// TIA Portal project "paletizer_2026_03_07" (V18)
// Vorlageprojekt für das Buch mit Zielsystem S7-1200

(* hardware
DEVICE "S7-1200 station_1"  S7-1200 Station
   slot 0: "Rack_0"  S7-1200 Rack  Rack  V1.0
   slot 1: "PLC_2"  CPU 1215C DC/DC/DC  6ES7 215-1AG40-0XB0  V4.4
   slot 2: "DI 16/DQ 16x24VDC_1"  6ES7 223-1BL32-0XB0  V2.0
   slot 3: "DI 16x24VDC_1"  6ES7 221-1BH32-0XB0  V2.0
   slot 4: "AI 4x13BIT/AQ 2x14BIT_1"  6ES7 234-4HE32-0XB0  V2.1
DEVICE "HMI_1"  KTP1200 Basic PN
   slot 0: "HMI_1"  KTP1200 Basic PN  6AV2 123-2MB03-0AX0  17.0.0.0
   slot 1: "HMI_RT_1"  KTP1200 Basic PN  6AV2 123-2MB03-0AX0  17.0.0.0
   slot 5: "HMI_1.IE_CP_1"  PROFINET Interface  17.0.0.0
      slot 1: "PROFINET Interface_1"  PROFINET Interface
         slot 1: "Port_1"  Port
*)

// ===== PLC "PLC_2"  CPU 1215C DC/DC/DC =====

VAR_GLOBAL   // PLC tag table "Default tag table"
   "Security Relay" AT %I10.0 : Bool;
   "Emergency stop feeding" AT %I10.1 : Bool;
   "Emergency stop elevator" AT %I10.2 : Bool;
   "Emergency stop load beld" AT %I10.3 : Bool;
   "Select auto" AT %I10.4 : Bool;
   "Select manual" AT %I10.5 : Bool;
   "Fault reset button" AT %I10.6 : Bool;
   "Manual box feeding button" AT %I11.0 : Bool;
   "Manual load beld" AT %I11.1 : Bool;
   "Manual Clamp" AT %I11.2 : Bool;
   "Box feeder motor guard" AT %I12.0 : Bool;
   "Enable load beld motor guard" AT %I12.1 : Bool;
   "Elevator motor guard" AT %I12.2 : Bool;
   "Load pallet motor guard" AT %I12.3 : Bool;
   "Pallet feeder motor guard" AT %I12.4 : Bool;
   "Exit conveyor motor guard" AT %I12.5 : Bool;
   "Box feeder motor feedback" AT %I13.0 : Bool;
   "Enable load beld motor feedback" AT %I13.1 : Bool;
   "Elevator motor feedback up" AT %I13.2 : Bool;
   "Elevator motor feedback down" AT %I13.3 : Bool;
   "Load pallet motor feedback" AT %I13.4 : Bool;
   "Pallet feeder motor feedback" AT %I13.5 : Bool;
   "Exit conveyor motor feedback" AT %I13.6 : Bool;
   "Pallet at entry" AT %I14.0 : Bool;
   "Pallet at exit" AT %I14.1 : Bool;
   "Pallet loaded" AT %I14.2 : Bool;
   "Up load pallet" AT %I14.3 : Bool;
   "Down load pallet" AT %I14.4 : Bool;
   "Box at entry" AT %I14.5 : Bool;
   "Pusher limit" AT %I14.6 : Bool;
   "Plate limit" AT %I14.7 : Bool;
   "Clamped" AT %I15.0 : Bool;
   "Manual pallet feeder" AT %I11.3 : Bool;
   "Manual load pallet" AT %I11.4 : Bool;
   "Elevator moving" AT %I15.1 : Bool;
   "Manual exit conveyor" AT %I11.5 : Bool;
   "Manual elevator up" AT %I15.2 : Bool;
   "Manual elevator down" AT %I15.3 : Bool;
   "Relay warning ligth" AT %Q10.0 : Bool;
   "Relay aux turn valve" AT %Q10.1 : Bool;
   "Relay aux push valve" AT %Q10.2 : Bool;
   "Relay aux plate valve" AT %Q10.3 : Bool;
   "Relay Clamp" AT %Q10.4 : Bool;
   "Move to limit" AT %Q10.5 : Bool;
   "Enable pallet emiter" AT %Q10.6 : Bool;
   "Enable exit conveyor" AT %Q10.7 : Bool;
   "Enable box feeder motor" AT %Q12.0 : Bool;
   "Enable load beld motor" AT %Q12.1 : Bool;
   "Enable elevator up motor" AT %Q12.2 : Bool;
   "Enable elevator down motor" AT %Q12.3 : Bool;
   "Enable Load pallet motor" AT %Q12.4 : Bool;
   "Enable Pallet feeder motor" AT %Q12.5 : Bool;
   "Enable exit conveyor motor" AT %Q12.6 : Bool;
   "Fault reset light" AT %Q13.0 : Bool;
   "Start feeding light" AT %Q13.1 : Bool;
   "Stop feeding light" AT %Q13.2 : Bool;
   "Counter box" AT %QW50 : Word;
   "Input_Security_Relay" AT %M0.0 : Bool;
   "Input_Emergency_stop_feeding" AT %M0.1 : Bool;
   "Input_emergency_stop_elevator" AT %M0.2 : Bool;
   "Input_emergency_stop_load_beld" AT %M0.3 : Bool;
   "Input_select_auto" AT %M0.4 : Bool;
   "Input_select_manual" AT %M0.5 : Bool;
   "Input_Fault_reset_button" AT %M0.6 : Bool;
   "Input_manual_box_feeding_button" AT %M1.0 : Bool;
   "Input_manual_load_beld" AT %M1.1 : Bool;
   "Input_manual_clamp" AT %M1.2 : Bool;
   "Input_manual_pallet_feeder" AT %M1.3 : Bool;
   "Input_box_feeder_motor_guard" AT %M2.0 : Bool;
   "Input_enable_load_beld_motor_guard" AT %M2.1 : Bool;
   "Input_elevator_motor_guard" AT %M2.2 : Bool;
   "Input_load_pallet_motor_guard" AT %M2.3 : Bool;
   "Input_pallet_feeder_motor_guad" AT %M2.4 : Bool;
   "Input_box_feeder_motor_feedback" AT %M3.0 : Bool;
   "Input_enable_load_beld_motor_feedback" AT %M3.1 : Bool;
   "Input_elevator_motor_feedback_up" AT %M3.2 : Bool;
   "Input_elevator_motor_feedback_down" AT %M3.3 : Bool;
   "Input_load_pallet_motor_feedback" AT %M3.4 : Bool;
   "Input_pallet_feeder_motor_feedback" AT %M3.5 : Bool;
   "Input_pallet_at_entry" AT %M4.0 : Bool;
   "Input_pallet_at_exit" AT %M4.1 : Bool;
   "Input_pallet_loaded" AT %M4.2 : Bool;
   "Input_up_load_pallet" AT %M4.3 : Bool;
   "Input_down_load_pallet" AT %M4.4 : Bool;
   "Input_box_at_entry" AT %M4.5 : Bool;
   "Input_pusher_limit" AT %M4.6 : Bool;
   "Input_plate_limit" AT %M4.7 : Bool;
   "Input_clamped" AT %M5.0 : Bool;
   "Output_warning_ligth" AT %M10.0 : Bool;
   "Output_relay_aux_turn_valve" AT %M10.1 : Bool;
   "Ouput_relay_aux_push_valve" AT %M10.2 : Bool;
   "Output_relay_aux_plate_valve" AT %M10.3 : Bool;
   "Output_relay_clamp" AT %M10.4 : Bool;
   "Ouput_move_to_limit" AT %M10.5 : Bool;
   "Output_enable_pallet_emiter" AT %M10.6 : Bool;
   "Output_enable_exit_conveyor" AT %M10.7 : Bool;
   "Output_enable_box_feeder_motor" AT %M12.0 : Bool;
   "Output_enable_load_beld_motor" AT %M12.1 : Bool;
   "Output_enable_elevator_up_motor" AT %M12.2 : Bool;
   "Output_enable_elevator_down_motor" AT %M12.3 : Bool;
   "Output_enable_load_pallet_motor" AT %M12.4 : Bool;
   "Output_enable_pallet_feeder_motor" AT %M12.5 : Bool;
   "Output_enable_exit_conveyor_motor" AT %M12.6 : Bool;
   "Output_fault_reset_light" AT %M13.0 : Bool;
   "Output_start_feeding_light" AT %M13.1 : Bool;
   "Output_stop_feeding_light" AT %M13.2 : Bool;
   "Ouput_counter_box" AT %MW100 : Word;
   "Emergency_enable" AT %M30.0 : Bool;
   "Manual_box_feeding_drive" AT %M30.1 : Bool;
   "Input_manual_load_pallet" AT %M1.4 : Bool;
   "Input_manual_exit_conveyor" AT %M1.5 : Bool;
   "Manual_load_beld_drive" AT %M30.2 : Bool;
   "Manual_clamp_drive" AT %M30.3 : Bool;
   "Manual_pallet_feeder_drive" AT %M30.4 : Bool;
   "Input_elevator_moving" AT %M5.1 : Bool;
   "Input_manual_elevator_up" AT %M5.2 : Bool;
   "Input_manual_elevator_down" AT %M5.3 : Bool;
   "Manual_load_pallet_drive" AT %M30.5 : Bool;
   "Manual_exit_conveyor_drive" AT %M30.6 : Bool;
   "Manual_elevator_up_drive" AT %M30.7 : Bool;
   "Manual_elevator_down_drive" AT %M31.0 : Bool;
   "Input_exit_conveyor_motor_guard" AT %M2.5 : Bool;
   "Input_exit_conveyor_motor_feedback" AT %M3.6 : Bool;
   "Aux_manual_box_feeding_drive" AT %M31.1 : Bool;
   "Up_manual_box_feeding_drive" AT %M6.0 : Bool;
   "Up_manual_load_beld_drive" AT %M6.1 : Bool;
   "Aux_manual_load_beld_drive" AT %M31.2 : Bool;
   "Aux_manual_pallet_feeder_drive" AT %M31.4 : Bool;
   "Aux_manual_load_pallet_drive" AT %M31.5 : Bool;
   "Aux_manual_exit_conveyor_drive" AT %M31.6 : Bool;
   "Aux_manual_elevator_up_drive" AT %M31.7 : Bool;
   "Aux_manual_elevator_down_drive" AT %M32.0 : Bool;
   "Up_manual_pallet_feeder_drive" AT %M6.2 : Bool;
   "Up_manual_load_pallet_drive" AT %M6.3 : Bool;
   "Up_manual_exit_conveyor_drive" AT %M6.4 : Bool;
   "Up_manual_elevator_up_drive" AT %M6.5 : Bool;
   "Up_manual_elevator_down_drive" AT %M6.6 : Bool;
   "Zero_Point" AT %M15.0 : Bool;
   "Reset_value_counters" AT %M15.2 : Bool;
   "Enable_Box_Feeder_Auto" AT %M15.3 : Bool;
   "Enable_Turn_Auto" AT %M15.4 : Bool;
   "Enable_Load_Beld_Auto" AT %M15.5 : Bool;
   "Enable_Push_Auto" AT %M15.6 : Bool;
   "Up_timer_0" AT %M50.0 : Bool;
   "Set_Counter_One" AT %M15.7 : Bool;
   "Up_Counter_one" AT %M50.1 : Bool;
   "Up_Counter_Two" AT %M50.2 : Bool;
   "Set_Counter_Two" AT %M16.0 : Bool;
   "Up_Counter_Three" AT %M50.3 : Bool;
   "Set_counter_Three" AT %M16.1 : Bool;
   "Up_Counter_Turn_Off_Two" AT %M50.4 : Bool;
   "Set_Counter_Five" AT %M16.2 : Bool;
   "Up_timer_3" AT %M50.5 : Bool;
   "Up_Zero_Point" AT %M50.6 : Bool;
   "Up_Set_Counter_Tur_Two" AT %M50.7 : Bool;
   "Up_Set_Counter_One" AT %M51.0 : Bool;
   "Up_Set_Counter_Two" AT %M51.1 : Bool;
   "Disable_Turn" AT %M16.3 : Bool;
   "Enable_Clamp_Auto" AT %M16.4 : Bool;
   "Up_Set_Counter_Turn" AT %M51.3 : Bool;
   "Up_Pusher_Limit" AT %M51.4 : Bool;
   "Prepare_Dish" AT %M16.5 : Bool;
   "Enable_Plate_Auto" AT %M16.6 : Bool;
   "Enable_Down_Elevator_Auto" AT %M16.7 : Bool;
   "Up_Input_clamped" AT %M51.5 : Bool;
   "Set_Counter_Four" AT %M17.0 : Bool;
   "Up_Counter_Turn_Two_Two" AT %M51.6 : Bool;
   "disable_pallet_loaded" AT %M17.1 : Bool;
   "enable_exit_conveyor_auto" AT %M17.2 : Bool;
   "turn_enable" AT %M17.3 : Bool;
   "Enable_feeder_pallet_auto" AT %M17.4 : Bool;
   "Enable_load_pallet_auto" AT %M17.5 : Bool;
   "Enable_Up_elevator_auto" AT %M17.6 : Bool;
   "Manual_turn_drive" AT %M17.7 : Bool;
   "Manual_plate_drive" AT %M18.0 : Bool;
   "Manual_push_drive" AT %M18.1 : Bool;
   "Zero_point_" AT %M51.7 : Bool;
   "Set_litter_value" AT %M18.2 : Bool;
   "Set_box_value" AT %M18.3 : Bool;
END_VAR

DATA_BLOCK "Engine_starter_DB_box_feeder"   // DB1
{ S7_Optimized_Access := 'TRUE' }
VERSION : 0.1
// stored: InstanceOfName Engine_starter
"Engine_starter"
BEGIN
END_DATA_BLOCK

DATA_BLOCK "Engine_starter_DB_load_beld"   // DB2
{ S7_Optimized_Access := 'TRUE' }
VERSION : 0.1
// stored: InstanceOfName Engine_starter
"Engine_starter"
BEGIN
END_DATA_BLOCK

DATA_BLOCK "Engine_starter_DB_elevator_up"   // DB3
{ S7_Optimized_Access := 'TRUE' }
VERSION : 0.1
// stored: InstanceOfName Engine_starter
"Engine_starter"
BEGIN
END_DATA_BLOCK

DATA_BLOCK "Engine_starter_DB_elevator_down"   // DB4
{ S7_Optimized_Access := 'TRUE' }
VERSION : 0.1
// stored: InstanceOfName Engine_starter
"Engine_starter"
BEGIN
END_DATA_BLOCK

DATA_BLOCK "Engine_starter_DB_load_pallet"   // DB5
{ S7_Optimized_Access := 'TRUE' }
VERSION : 0.1
// stored: InstanceOfName Engine_starter
"Engine_starter"
BEGIN
END_DATA_BLOCK

DATA_BLOCK "Engine_starter_DB_pallet_feeder"   // DB6
{ S7_Optimized_Access := 'TRUE' }
VERSION : 0.1
// stored: InstanceOfName Engine_starter
"Engine_starter"
BEGIN
END_DATA_BLOCK

DATA_BLOCK "Engine_starter_DB_exit_conveyor"   // DB7
{ S7_Optimized_Access := 'TRUE' }
VERSION : 0.1
// stored: InstanceOfName Engine_starter
"Engine_starter"
BEGIN
END_DATA_BLOCK

DATA_BLOCK "HMI"   // DB28
{ S7_Optimized_Access := 'FALSE' }
VERSION : 0.1
   VAR
      Mode_manual : Bool;
      Mode_auto : Bool;
      Mode_manual_actived : Bool;
      Mode_auto_actived : Bool;
      Mode_rest : Bool;
      Reset : Bool;
      List_status : Int;
      Start_box_feeder : Bool;
      Stop_box_feeder : Bool;
      Enable_box_feeder : Bool;
      Enabled_box_feeder : Bool;
      Failure_active_emergency_box_feeder : Bool;
      Failure_active_thermal_box_feeder : Bool;
      Failure_feedback_box_feeder : Bool;
      Failure_box_feeder : Bool;
      Status_box_feeder : Int;
      List_failure_box_feeder : Int;
      Rotation_box_feeder : Int;
      Start_load_beld : Bool;
      Stop_load_beld : Bool;
      Enable_load_beld : Bool;
      Enabled_load_beld : Bool;
      Failure_active_emergency_load_beld : Bool;
      Failure_active_thermal_load_beld : Bool;
      Failure_feedback_load_beld : Bool;
      Failure_load_beld : Bool;
      Status_load_beld : Int;
      List_failure_load_beld : Int;
      Rotation_load_beld : Int;
      Up_elevator : Bool;
      Down_elevator : Bool;
      Enable_up_elevator : Bool;
      Enable_down_elevator : Bool;
      Enabled_up_elevator : Bool;
      Enabled_down_elevator : Bool;
      Enabled_elevator : Bool;
      Failure_active_emergency_elevator : Bool;
      Failure_active_thermal_elevator : Bool;
      Failure_feedback_elevator : Bool;
      Failure_elevator : Bool;
      Status_elevator : Int;
      List_failure_elevator : Int;
      Rotation_elevator : Int;
      Start_load_pallet : Bool;
      Stop_load_pallet : Bool;
      Enable_load_pallet : Bool;
      Enabled_load_pallet : Bool;
      Failure_active_emergency_load_pallet : Bool;
      Failure_active_thermal_load_pallet : Bool;
      Failure_feedback_load_pallet : Bool;
      Failure_load_pallet : Bool;
      Status_load_pallet : Int;
      List_failure_load_pallet : Int;
      Rotation_load_pallet : Int;
      Start_pallet_feeder : Bool;
      Stop_pallet_feeder : Bool;
      Enable_pallet_feeder : Bool;
      Enabled_pallet_feeder : Bool;
      Failure_active_emergency_pallet_feeder : Bool;
      Failure_active_thermal_pallet_feeder : Bool;
      Failure_feedback_pallet_feeder : Bool;
      Failure_pallet_feeder : Bool;
      Status_pallet_feeder : Int;
      List_failure_pallet_feeder : Int;
      Rotation_pallet_feeder : Int;
      Start_exit_conveyor : Bool;
      Stop_exit_conveyor : Bool;
      Enable_exit_conveyor : Bool;
      Enabled_exit_conveyor : Bool;
      Failure_active_emergency_exit_conveyor : Bool;
      Failure_active_thermal_exit_conveyor : Bool;
      Failure_feedback_exit_conveyor : Bool;
      Failure_exit_conveyor : Bool;
      Status_exit_conveyor : Int;
      List_failure_exit_conveyor : Int;
      Rotation_exit_conveyor : Int;
      Enable_turn : Bool;
      Enabled_turn : Bool;
      Enable_push : Bool;
      Enabled_push : Bool;
      Enable_plate : Bool;
      Enabled_plate : Bool;
      Enable_clamp : Bool;
      Enabled_clamp : Bool;
      Box_counter : Bool;
      cero_point : Bool;
      Elevator_moving : Int;
      Set_box : Int;
      Set_litter : Int;
      Box_input_counter : Int;
      Completed_pallets_counter : Int;
      List_failure_and_warning : Int;
   END_VAR
BEGIN
END_DATA_BLOCK

DATA_BLOCK "HMI_motor_rotation_box_feeder"   // DB32
{ S7_Optimized_Access := 'TRUE' }
VERSION : 0.1
// stored: InstanceOfName HMI_motor_rotation
"HMI_motor_rotation"
BEGIN
END_DATA_BLOCK

DATA_BLOCK "HMI_motor_rotation_load_beld"   // DB33
{ S7_Optimized_Access := 'TRUE' }
VERSION : 0.1
// stored: InstanceOfName HMI_motor_rotation
"HMI_motor_rotation"
BEGIN
END_DATA_BLOCK

DATA_BLOCK "HMI_motor_rotation_elevator"   // DB34
{ S7_Optimized_Access := 'TRUE' }
VERSION : 0.1
// stored: InstanceOfName HMI_motor_rotation
"HMI_motor_rotation"
BEGIN
END_DATA_BLOCK

DATA_BLOCK "HMI_motor_rotation_load_pallet"   // DB35
{ S7_Optimized_Access := 'TRUE' }
VERSION : 0.1
// stored: InstanceOfName HMI_motor_rotation
"HMI_motor_rotation"
BEGIN
END_DATA_BLOCK

DATA_BLOCK "HMI_motor_rotation_pallet_feeder"   // DB36
{ S7_Optimized_Access := 'TRUE' }
VERSION : 0.1
// stored: InstanceOfName HMI_motor_rotation
"HMI_motor_rotation"
BEGIN
END_DATA_BLOCK

DATA_BLOCK "HMI_motor_rotation_exit_conveyor"   // DB37
{ S7_Optimized_Access := 'TRUE' }
VERSION : 0.1
// stored: InstanceOfName HMI_motor_rotation
"HMI_motor_rotation"
BEGIN
END_DATA_BLOCK

// folder: System blocks/Program resources

DATA_BLOCK "Counter_one"   // DB8
{ S7_Optimized_Access := 'TRUE' }
AUTHOR : Simatic
FAMILY : IEC
NAME : CNTR
VERSION : 1.0
// stored: InstanceOfName IEC_COUNTER
"IEC_COUNTER"
BEGIN
END_DATA_BLOCK

DATA_BLOCK "Counter_two"   // DB9
{ S7_Optimized_Access := 'TRUE' }
AUTHOR : Simatic
FAMILY : IEC
NAME : CNTR
VERSION : 1.0
// stored: InstanceOfName IEC_COUNTER
"IEC_COUNTER"
BEGIN
END_DATA_BLOCK

DATA_BLOCK "Counter_Three"   // DB10
{ S7_Optimized_Access := 'TRUE' }
AUTHOR : Simatic
FAMILY : IEC
NAME : CNTR
VERSION : 1.0
// stored: InstanceOfName IEC_COUNTER
"IEC_COUNTER"
BEGIN
END_DATA_BLOCK

DATA_BLOCK "Counter_five"   // DB11
{ S7_Optimized_Access := 'TRUE' }
AUTHOR : Simatic
FAMILY : IEC
NAME : CNTR
VERSION : 1.0
// stored: InstanceOfName IEC_COUNTER
"IEC_COUNTER"
BEGIN
END_DATA_BLOCK

DATA_BLOCK "Timer_0"   // DB12
{ S7_Optimized_Access := 'TRUE' }
AUTHOR : Simatic
FAMILY : IEC
NAME : IEC_TMR
VERSION : 1.0
// stored: InstanceOfName IEC_TIMER
"IEC_TIMER"
BEGIN
END_DATA_BLOCK

DATA_BLOCK "Timer_1"   // DB13
{ S7_Optimized_Access := 'TRUE' }
AUTHOR : Simatic
FAMILY : IEC
NAME : IEC_TMR
VERSION : 1.0
// stored: InstanceOfName IEC_TIMER
"IEC_TIMER"
BEGIN
END_DATA_BLOCK

DATA_BLOCK "Timer_3"   // DB14
{ S7_Optimized_Access := 'TRUE' }
AUTHOR : Simatic
FAMILY : IEC
NAME : IEC_TMR
VERSION : 1.0
// stored: InstanceOfName IEC_TIMER
"IEC_TIMER"
BEGIN
END_DATA_BLOCK

DATA_BLOCK "time_4"   // DB15
{ S7_Optimized_Access := 'TRUE' }
AUTHOR : Simatic
FAMILY : IEC
NAME : IEC_TMR
VERSION : 1.0
// stored: InstanceOfName IEC_TIMER
"IEC_TIMER"
BEGIN
END_DATA_BLOCK

DATA_BLOCK "Timer_4"   // DB16
{ S7_Optimized_Access := 'TRUE' }
AUTHOR : Simatic
FAMILY : IEC
NAME : IEC_TMR
VERSION : 1.0
// stored: InstanceOfName IEC_TIMER
"IEC_TIMER"
BEGIN
END_DATA_BLOCK

DATA_BLOCK "Timer_19"   // DB17
{ S7_Optimized_Access := 'TRUE' }
AUTHOR : Simatic
FAMILY : IEC
NAME : IEC_TMR
VERSION : 1.0
// stored: InstanceOfName IEC_TIMER
"IEC_TIMER"
BEGIN
END_DATA_BLOCK

DATA_BLOCK "Timer_16"   // DB18
{ S7_Optimized_Access := 'TRUE' }
AUTHOR : Simatic
FAMILY : IEC
NAME : IEC_TMR
VERSION : 1.0
// stored: InstanceOfName IEC_TIMER
"IEC_TIMER"
BEGIN
END_DATA_BLOCK

DATA_BLOCK "Timer_7"   // DB19
{ S7_Optimized_Access := 'TRUE' }
AUTHOR : Simatic
FAMILY : IEC
NAME : IEC_TMR
VERSION : 1.0
// stored: InstanceOfName IEC_TIMER
"IEC_TIMER"
BEGIN
END_DATA_BLOCK

DATA_BLOCK "Timer_8"   // DB20
{ S7_Optimized_Access := 'TRUE' }
AUTHOR : Simatic
FAMILY : IEC
NAME : IEC_TMR
VERSION : 1.0
// stored: InstanceOfName IEC_TIMER
"IEC_TIMER"
BEGIN
END_DATA_BLOCK

DATA_BLOCK "Timer_9"   // DB21
{ S7_Optimized_Access := 'TRUE' }
AUTHOR : Simatic
FAMILY : IEC
NAME : IEC_TMR
VERSION : 1.0
// stored: InstanceOfName IEC_TIMER
"IEC_TIMER"
BEGIN
END_DATA_BLOCK

DATA_BLOCK "Timer_off_one"   // DB22
{ S7_Optimized_Access := 'TRUE' }
AUTHOR : Simatic
FAMILY : IEC
NAME : IEC_TMR
VERSION : 1.0
// stored: InstanceOfName IEC_TIMER
"IEC_TIMER"
BEGIN
END_DATA_BLOCK

DATA_BLOCK "Litter_counter"   // DB23
{ S7_Optimized_Access := 'TRUE' }
AUTHOR : Simatic
FAMILY : IEC
NAME : CNTR
VERSION : 1.0
// stored: InstanceOfName IEC_COUNTER
"IEC_COUNTER"
BEGIN
END_DATA_BLOCK

DATA_BLOCK "Timer_10"   // DB24
{ S7_Optimized_Access := 'TRUE' }
AUTHOR : Simatic
FAMILY : IEC
NAME : IEC_TMR
VERSION : 1.0
// stored: InstanceOfName IEC_TIMER
"IEC_TIMER"
BEGIN
END_DATA_BLOCK

DATA_BLOCK "Timer_11"   // DB25
{ S7_Optimized_Access := 'TRUE' }
AUTHOR : Simatic
FAMILY : IEC
NAME : IEC_TMR
VERSION : 1.0
// stored: InstanceOfName IEC_TIMER
"IEC_TIMER"
BEGIN
END_DATA_BLOCK

DATA_BLOCK "Counter_four"   // DB26
{ S7_Optimized_Access := 'TRUE' }
AUTHOR : Simatic
FAMILY : IEC
NAME : CNTR
VERSION : 1.0
// stored: InstanceOfName IEC_COUNTER
"IEC_COUNTER"
BEGIN
END_DATA_BLOCK

DATA_BLOCK "Timer_12"   // DB27
{ S7_Optimized_Access := 'TRUE' }
AUTHOR : Simatic
FAMILY : IEC
NAME : IEC_TMR
VERSION : 1.0
// stored: InstanceOfName IEC_TIMER
"IEC_TIMER"
BEGIN
END_DATA_BLOCK

DATA_BLOCK "timer_13"   // DB29
{ S7_Optimized_Access := 'TRUE' }
AUTHOR : Simatic
FAMILY : IEC
NAME : IEC_TMR
VERSION : 1.0
// stored: InstanceOfName IEC_TIMER
"IEC_TIMER"
BEGIN
END_DATA_BLOCK

DATA_BLOCK "Timer_14"   // DB30
{ S7_Optimized_Access := 'TRUE' }
AUTHOR : Simatic
FAMILY : IEC
NAME : IEC_TMR
VERSION : 1.0
// stored: InstanceOfName IEC_TIMER
"IEC_TIMER"
BEGIN
END_DATA_BLOCK

DATA_BLOCK "Timer_15"   // DB31
{ S7_Optimized_Access := 'TRUE' }
AUTHOR : Simatic
FAMILY : IEC
NAME : IEC_TMR
VERSION : 1.0
// stored: InstanceOfName IEC_TIMER
"IEC_TIMER"
BEGIN
END_DATA_BLOCK

DATA_BLOCK "Box_input_counter"   // DB38
{ S7_Optimized_Access := 'TRUE' }
AUTHOR : Simatic
FAMILY : IEC
NAME : CNTR
VERSION : 1.0
// stored: InstanceOfName IEC_COUNTER
"IEC_COUNTER"
BEGIN
END_DATA_BLOCK

DATA_BLOCK "litter_counter_display"   // DB39
{ S7_Optimized_Access := 'TRUE' }
AUTHOR : Simatic
FAMILY : IEC
NAME : CNTR
VERSION : 1.0
// stored: InstanceOfName IEC_COUNTER
"IEC_COUNTER"
BEGIN
END_DATA_BLOCK

// folder: (top level)

FUNCTION_BLOCK "Engine_starter"   // FB1, LAD
{ S7_Optimized_Access := 'TRUE' }
VERSION : 0.1
   VAR_INPUT
      STOP_EMERGENCY : Bool;
      THERMAL_SHUTDOWN : Bool;
      CONTACT_FEEDBACK : Bool;
      ENABLE : Bool;
      RESET_FAULT : Bool;
      STOP_AUX : Bool;
   END_VAR
   VAR_OUTPUT
      START_ENABLED : Bool;
      STARTING_FAILURE : Bool;
      ACTIVE_EMERGENCY : Bool;
      ACTIVE_THERMAL : Bool;
      FEEDBACK_FAILURE : Bool;
   END_VAR
   VAR
      stop_error : Bool;
      temp_feedback : TON_TIME;
      enable_engine : Bool;
      temp_thermal_shutdown : TON_TIME;
   END_VAR
BEGIN

REGION Network 1
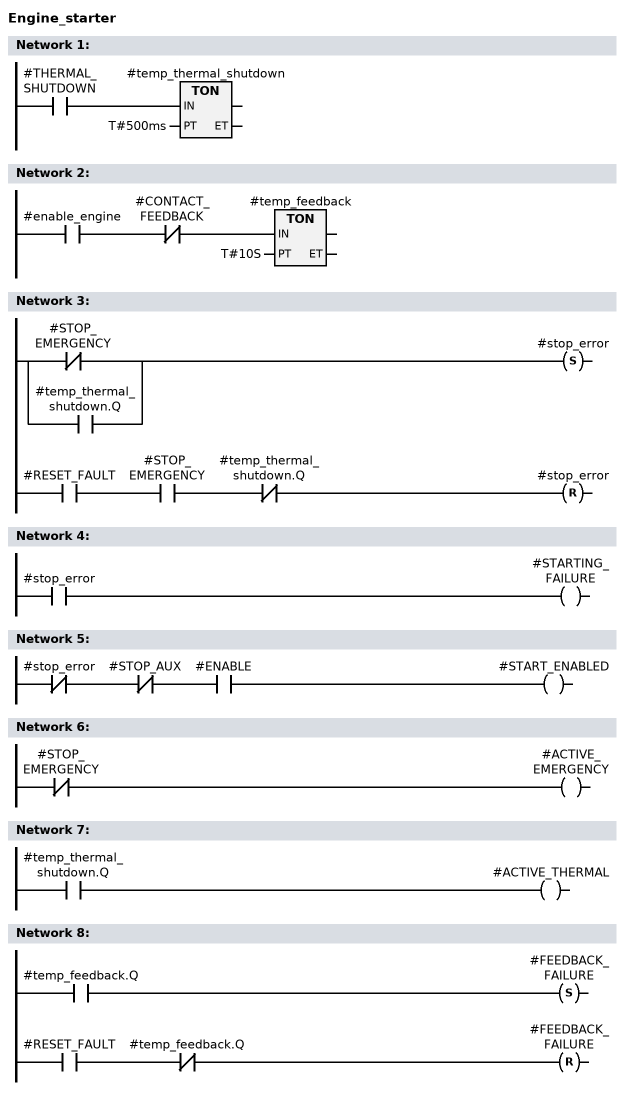
   #temp_thermal_shutdown(IN := #THERMAL_SHUTDOWN, PT := T#500ms);   // TON
END_REGION

REGION Network 2
   #temp_feedback(IN := #enable_engine AND NOT #CONTACT_FEEDBACK, PT := T#10S);   // TON
END_REGION

REGION Network 3
   RUNG wire#powerrail
      I_Contact( #STOP_EMERGENCY )
      wire#w1
      S_Coil( #stop_error )
   END_RUNG
   RUNG wire#powerrail
      Contact( #temp_thermal_shutdown.Q )
   END_RUNG wire#w1
   RUNG wire#powerrail
      Contact( #RESET_FAULT )
      Contact( #STOP_EMERGENCY )
      I_Contact( #temp_thermal_shutdown.Q )
      R_Coil( #stop_error )
   END_RUNG
   // the same network as SCL:
   IF NOT #STOP_EMERGENCY OR #temp_thermal_shutdown.Q THEN #stop_error := TRUE; END_IF;
   IF #RESET_FAULT AND #STOP_EMERGENCY AND NOT #temp_thermal_shutdown.Q THEN #stop_error := FALSE; END_IF;
END_REGION

REGION Network 4
   RUNG wire#powerrail
      Contact( #stop_error )
      Coil( #STARTING_FAILURE )
   END_RUNG
   // the same network as SCL:
   #STARTING_FAILURE := #stop_error;
END_REGION

REGION Network 5
   RUNG wire#powerrail
      I_Contact( #stop_error )
      I_Contact( #STOP_AUX )
      Contact( #ENABLE )
      Coil( #START_ENABLED )
   END_RUNG
   // the same network as SCL:
   #START_ENABLED := NOT #stop_error AND NOT #STOP_AUX AND #ENABLE;
END_REGION

REGION Network 6
   RUNG wire#powerrail
      I_Contact( #STOP_EMERGENCY )
      Coil( #ACTIVE_EMERGENCY )
   END_RUNG
   // the same network as SCL:
   #ACTIVE_EMERGENCY := NOT #STOP_EMERGENCY;
END_REGION

REGION Network 7
   RUNG wire#powerrail
      Contact( #temp_thermal_shutdown.Q )
      Coil( #ACTIVE_THERMAL )
   END_RUNG
   // the same network as SCL:
   #ACTIVE_THERMAL := #temp_thermal_shutdown.Q;
END_REGION

REGION Network 8
   RUNG wire#powerrail
      Contact( #temp_feedback.Q )
      S_Coil( #FEEDBACK_FAILURE )
   END_RUNG
   RUNG wire#powerrail
      Contact( #RESET_FAULT )
      I_Contact( #temp_feedback.Q )
      R_Coil( #FEEDBACK_FAILURE )
   END_RUNG
   // the same network as SCL:
   IF #temp_feedback.Q THEN #FEEDBACK_FAILURE := TRUE; END_IF;
   IF #RESET_FAULT AND NOT #temp_feedback.Q THEN #FEEDBACK_FAILURE := FALSE; END_IF;
END_REGION
END_FUNCTION_BLOCK

FUNCTION_BLOCK "HMI_motor_rotation"   // FB2, LAD
{ S7_Optimized_Access := 'TRUE' }
VERSION : 0.1
   VAR_INPUT
      enable_motor : Bool;
   END_VAR
   VAR_OUTPUT
      Motor_rotation : Int;
   END_VAR
   VAR
      time_one : TON_TIME;
      time_two : TON_TIME;
      time_three : TON_TIME;
      time_four : TON_TIME;
      time_five : TON_TIME;
   END_VAR
   VAR_TEMP   // added for the SCL form of the ladder/FBD networks
      _w1 : Bool;
   END_VAR
BEGIN

REGION Network 1
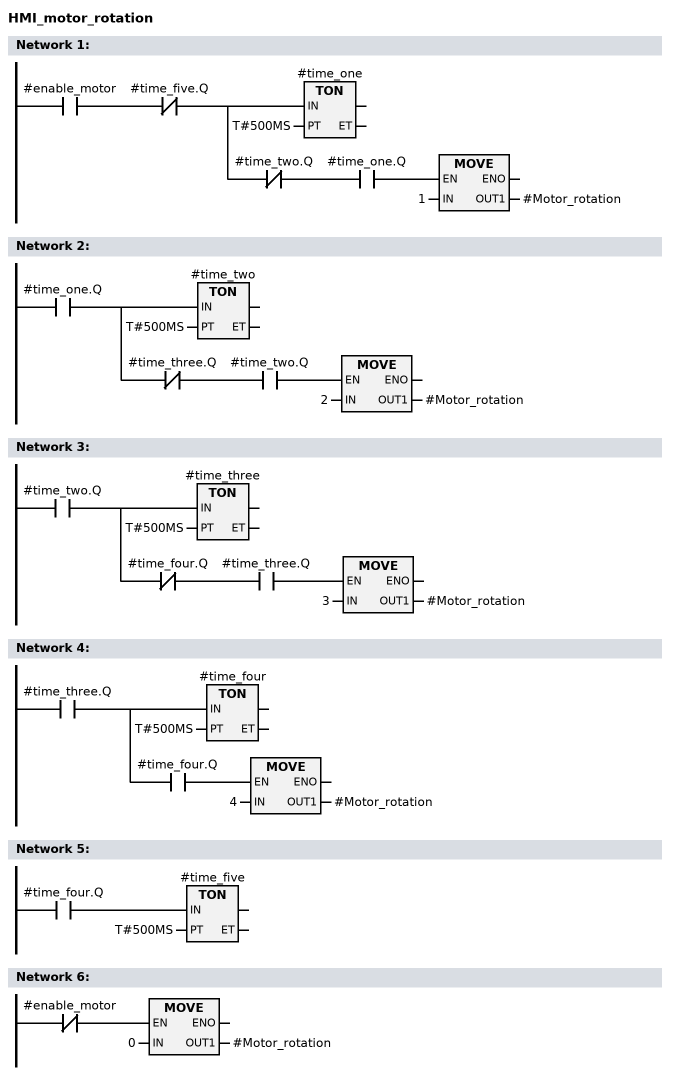
   #_w1 := #enable_motor AND NOT #time_five.Q;
   #time_one(IN := #_w1, PT := T#500MS);   // TON
   IF #_w1 AND NOT #time_two.Q AND #time_one.Q THEN #Motor_rotation := 1; END_IF;
END_REGION

REGION Network 2
   #time_two(IN := #time_one.Q, PT := T#500MS);   // TON
   IF #time_one.Q AND NOT #time_three.Q AND #time_two.Q THEN #Motor_rotation := 2; END_IF;
END_REGION

REGION Network 3
   #time_three(IN := #time_two.Q, PT := T#500MS);   // TON
   IF #time_two.Q AND NOT #time_four.Q AND #time_three.Q THEN #Motor_rotation := 3; END_IF;
END_REGION

REGION Network 4
   #time_four(IN := #time_three.Q, PT := T#500MS);   // TON
   IF #time_three.Q AND #time_four.Q THEN #Motor_rotation := 4; END_IF;
END_REGION

REGION Network 5
   #time_five(IN := #time_four.Q, PT := T#500MS);   // TON
END_REGION

REGION Network 6
   RUNG wire#powerrail
      I_Contact( #enable_motor )
      Move(in := 0, out1 => #Motor_rotation)
   END_RUNG
   // the same network as SCL:
   IF NOT #enable_motor THEN #Motor_rotation := 0; END_IF;
END_REGION
END_FUNCTION_BLOCK

FUNCTION "Input_Management" : Void   // FC1, LAD
{ S7_Optimized_Access := 'TRUE' }
VERSION : 0.1
BEGIN

REGION Network 1
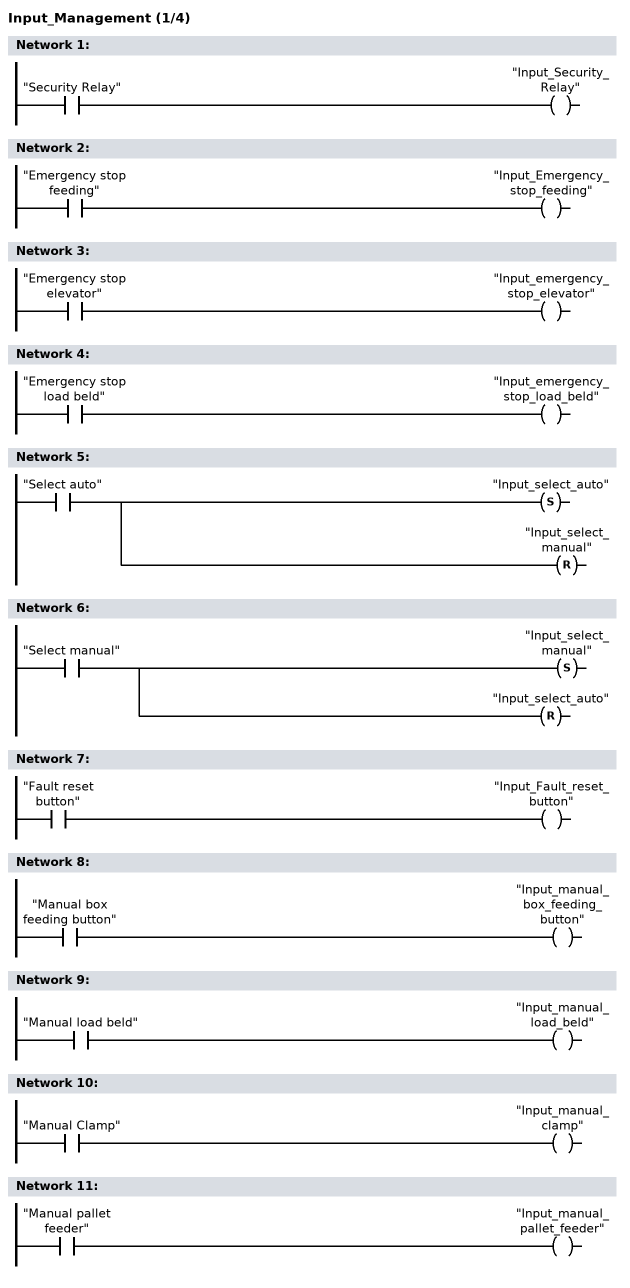
   RUNG wire#powerrail
      Contact( "Security Relay" )
      Coil( "Input_Security_Relay" )
   END_RUNG
   // the same network as SCL:
   "Input_Security_Relay" := "Security Relay";
END_REGION

REGION Network 2
   RUNG wire#powerrail
      Contact( "Emergency stop feeding" )
      Coil( "Input_Emergency_stop_feeding" )
   END_RUNG
   // the same network as SCL:
   "Input_Emergency_stop_feeding" := "Emergency stop feeding";
END_REGION

REGION Network 3
   RUNG wire#powerrail
      Contact( "Emergency stop elevator" )
      Coil( "Input_emergency_stop_elevator" )
   END_RUNG
   // the same network as SCL:
   "Input_emergency_stop_elevator" := "Emergency stop elevator";
END_REGION

REGION Network 4
   RUNG wire#powerrail
      Contact( "Emergency stop load beld" )
      Coil( "Input_emergency_stop_load_beld" )
   END_RUNG
   // the same network as SCL:
   "Input_emergency_stop_load_beld" := "Emergency stop load beld";
END_REGION

REGION Network 5
   RUNG wire#powerrail
      Contact( "Select auto" )
      wire#w1
      S_Coil( "Input_select_auto" )
   END_RUNG
   RUNG wire#w1
      R_Coil( "Input_select_manual" )
   END_RUNG
   // the same network as SCL:
   IF "Select auto" THEN
       "Input_select_auto" := TRUE;
       "Input_select_manual" := FALSE;
   END_IF;
END_REGION

REGION Network 6
   RUNG wire#powerrail
      Contact( "Select manual" )
      wire#w1
      S_Coil( "Input_select_manual" )
   END_RUNG
   RUNG wire#w1
      R_Coil( "Input_select_auto" )
   END_RUNG
   // the same network as SCL:
   IF "Select manual" THEN
       "Input_select_manual" := TRUE;
       "Input_select_auto" := FALSE;
   END_IF;
END_REGION

REGION Network 7
   RUNG wire#powerrail
      Contact( "Fault reset button" )
      Coil( "Input_Fault_reset_button" )
   END_RUNG
   // the same network as SCL:
   "Input_Fault_reset_button" := "Fault reset button";
END_REGION

REGION Network 8
   RUNG wire#powerrail
      Contact( "Manual box feeding button" )
      Coil( "Input_manual_box_feeding_button" )
   END_RUNG
   // the same network as SCL:
   "Input_manual_box_feeding_button" := "Manual box feeding button";
END_REGION

REGION Network 9
   RUNG wire#powerrail
      Contact( "Manual load beld" )
      Coil( "Input_manual_load_beld" )
   END_RUNG
   // the same network as SCL:
   "Input_manual_load_beld" := "Manual load beld";
END_REGION

REGION Network 10
   RUNG wire#powerrail
      Contact( "Manual Clamp" )
      Coil( "Input_manual_clamp" )
   END_RUNG
   // the same network as SCL:
   "Input_manual_clamp" := "Manual Clamp";
END_REGION

REGION Network 11
   RUNG wire#powerrail
      Contact( "Manual pallet feeder" )
      Coil( "Input_manual_pallet_feeder" )
   END_RUNG
   // the same network as SCL:
   "Input_manual_pallet_feeder" := "Manual pallet feeder";
END_REGION

REGION Network 12
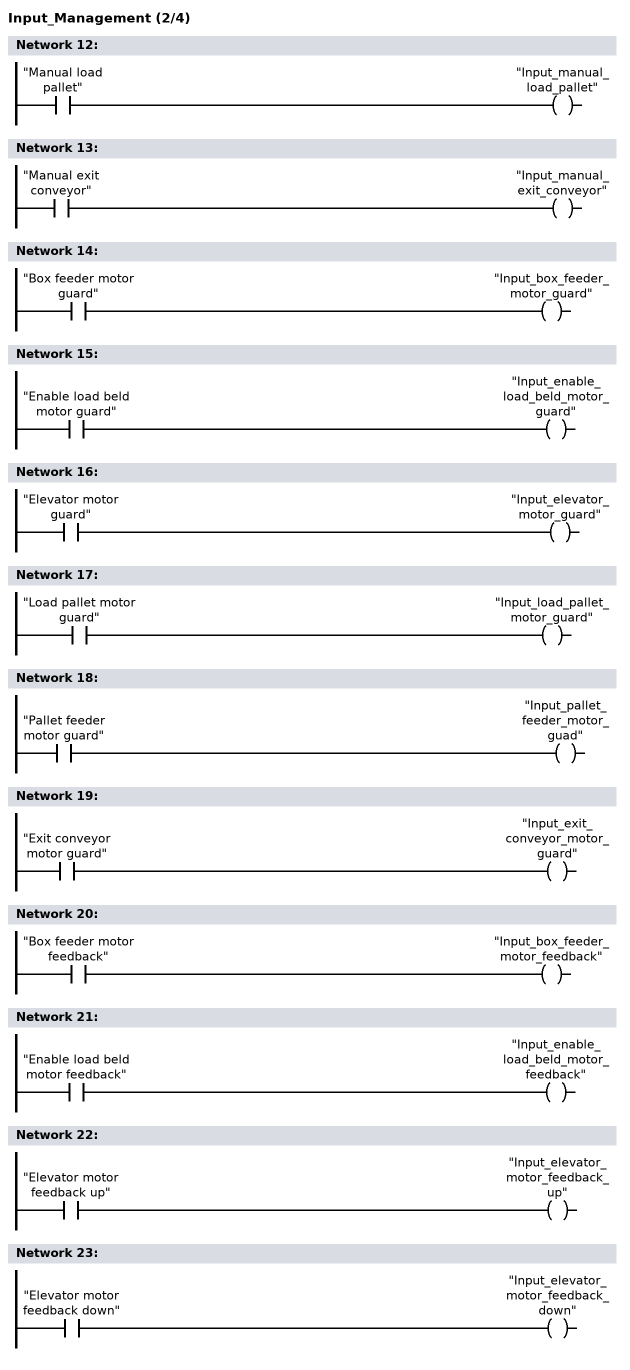
   RUNG wire#powerrail
      Contact( "Manual load pallet" )
      Coil( "Input_manual_load_pallet" )
   END_RUNG
   // the same network as SCL:
   "Input_manual_load_pallet" := "Manual load pallet";
END_REGION

REGION Network 13
   RUNG wire#powerrail
      Contact( "Manual exit conveyor" )
      Coil( "Input_manual_exit_conveyor" )
   END_RUNG
   // the same network as SCL:
   "Input_manual_exit_conveyor" := "Manual exit conveyor";
END_REGION

REGION Network 14
   RUNG wire#powerrail
      Contact( "Box feeder motor guard" )
      Coil( "Input_box_feeder_motor_guard" )
   END_RUNG
   // the same network as SCL:
   "Input_box_feeder_motor_guard" := "Box feeder motor guard";
END_REGION

REGION Network 15
   RUNG wire#powerrail
      Contact( "Enable load beld motor guard" )
      Coil( "Input_enable_load_beld_motor_guard" )
   END_RUNG
   // the same network as SCL:
   "Input_enable_load_beld_motor_guard" := "Enable load beld motor guard";
END_REGION

REGION Network 16
   RUNG wire#powerrail
      Contact( "Elevator motor guard" )
      Coil( "Input_elevator_motor_guard" )
   END_RUNG
   // the same network as SCL:
   "Input_elevator_motor_guard" := "Elevator motor guard";
END_REGION

REGION Network 17
   RUNG wire#powerrail
      Contact( "Load pallet motor guard" )
      Coil( "Input_load_pallet_motor_guard" )
   END_RUNG
   // the same network as SCL:
   "Input_load_pallet_motor_guard" := "Load pallet motor guard";
END_REGION

REGION Network 18
   RUNG wire#powerrail
      Contact( "Pallet feeder motor guard" )
      Coil( "Input_pallet_feeder_motor_guad" )
   END_RUNG
   // the same network as SCL:
   "Input_pallet_feeder_motor_guad" := "Pallet feeder motor guard";
END_REGION

REGION Network 19
   RUNG wire#powerrail
      Contact( "Exit conveyor motor guard" )
      Coil( "Input_exit_conveyor_motor_guard" )
   END_RUNG
   // the same network as SCL:
   "Input_exit_conveyor_motor_guard" := "Exit conveyor motor guard";
END_REGION

REGION Network 20
   RUNG wire#powerrail
      Contact( "Box feeder motor feedback" )
      Coil( "Input_box_feeder_motor_feedback" )
   END_RUNG
   // the same network as SCL:
   "Input_box_feeder_motor_feedback" := "Box feeder motor feedback";
END_REGION

REGION Network 21
   RUNG wire#powerrail
      Contact( "Enable load beld motor feedback" )
      Coil( "Input_enable_load_beld_motor_feedback" )
   END_RUNG
   // the same network as SCL:
   "Input_enable_load_beld_motor_feedback" := "Enable load beld motor feedback";
END_REGION

REGION Network 22
   RUNG wire#powerrail
      Contact( "Elevator motor feedback up" )
      Coil( "Input_elevator_motor_feedback_up" )
   END_RUNG
   // the same network as SCL:
   "Input_elevator_motor_feedback_up" := "Elevator motor feedback up";
END_REGION

REGION Network 23
   RUNG wire#powerrail
      Contact( "Elevator motor feedback down" )
      Coil( "Input_elevator_motor_feedback_down" )
   END_RUNG
   // the same network as SCL:
   "Input_elevator_motor_feedback_down" := "Elevator motor feedback down";
END_REGION

REGION Network 24
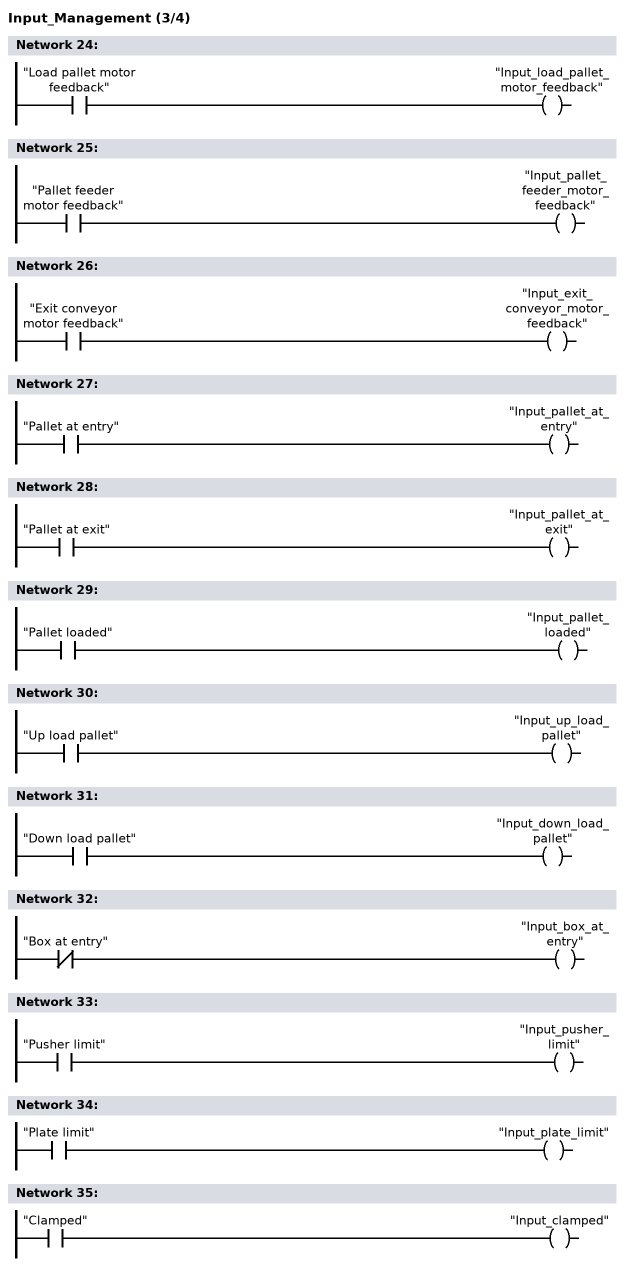
   RUNG wire#powerrail
      Contact( "Load pallet motor feedback" )
      Coil( "Input_load_pallet_motor_feedback" )
   END_RUNG
   // the same network as SCL:
   "Input_load_pallet_motor_feedback" := "Load pallet motor feedback";
END_REGION

REGION Network 25
   RUNG wire#powerrail
      Contact( "Pallet feeder motor feedback" )
      Coil( "Input_pallet_feeder_motor_feedback" )
   END_RUNG
   // the same network as SCL:
   "Input_pallet_feeder_motor_feedback" := "Pallet feeder motor feedback";
END_REGION

REGION Network 26
   RUNG wire#powerrail
      Contact( "Exit conveyor motor feedback" )
      Coil( "Input_exit_conveyor_motor_feedback" )
   END_RUNG
   // the same network as SCL:
   "Input_exit_conveyor_motor_feedback" := "Exit conveyor motor feedback";
END_REGION

REGION Network 27
   RUNG wire#powerrail
      Contact( "Pallet at entry" )
      Coil( "Input_pallet_at_entry" )
   END_RUNG
   // the same network as SCL:
   "Input_pallet_at_entry" := "Pallet at entry";
END_REGION

REGION Network 28
   RUNG wire#powerrail
      Contact( "Pallet at exit" )
      Coil( "Input_pallet_at_exit" )
   END_RUNG
   // the same network as SCL:
   "Input_pallet_at_exit" := "Pallet at exit";
END_REGION

REGION Network 29
   RUNG wire#powerrail
      Contact( "Pallet loaded" )
      Coil( "Input_pallet_loaded" )
   END_RUNG
   // the same network as SCL:
   "Input_pallet_loaded" := "Pallet loaded";
END_REGION

REGION Network 30
   RUNG wire#powerrail
      Contact( "Up load pallet" )
      Coil( "Input_up_load_pallet" )
   END_RUNG
   // the same network as SCL:
   "Input_up_load_pallet" := "Up load pallet";
END_REGION

REGION Network 31
   RUNG wire#powerrail
      Contact( "Down load pallet" )
      Coil( "Input_down_load_pallet" )
   END_RUNG
   // the same network as SCL:
   "Input_down_load_pallet" := "Down load pallet";
END_REGION

REGION Network 32
   RUNG wire#powerrail
      I_Contact( "Box at entry" )
      Coil( "Input_box_at_entry" )
   END_RUNG
   // the same network as SCL:
   "Input_box_at_entry" := NOT "Box at entry";
END_REGION

REGION Network 33
   RUNG wire#powerrail
      Contact( "Pusher limit" )
      Coil( "Input_pusher_limit" )
   END_RUNG
   // the same network as SCL:
   "Input_pusher_limit" := "Pusher limit";
END_REGION

REGION Network 34
   RUNG wire#powerrail
      Contact( "Plate limit" )
      Coil( "Input_plate_limit" )
   END_RUNG
   // the same network as SCL:
   "Input_plate_limit" := "Plate limit";
END_REGION

REGION Network 35
   RUNG wire#powerrail
      Contact( "Clamped" )
      Coil( "Input_clamped" )
   END_RUNG
   // the same network as SCL:
   "Input_clamped" := "Clamped";
END_REGION

REGION Network 36
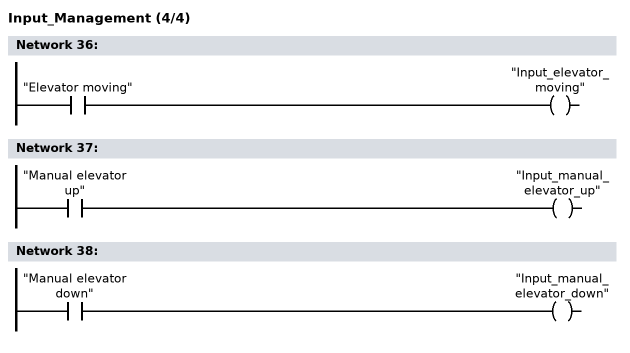
   RUNG wire#powerrail
      Contact( "Elevator moving" )
      Coil( "Input_elevator_moving" )
   END_RUNG
   // the same network as SCL:
   "Input_elevator_moving" := "Elevator moving";
END_REGION

REGION Network 37
   RUNG wire#powerrail
      Contact( "Manual elevator up" )
      Coil( "Input_manual_elevator_up" )
   END_RUNG
   // the same network as SCL:
   "Input_manual_elevator_up" := "Manual elevator up";
END_REGION

REGION Network 38
   RUNG wire#powerrail
      Contact( "Manual elevator down" )
      Coil( "Input_manual_elevator_down" )
   END_RUNG
   // the same network as SCL:
   "Input_manual_elevator_down" := "Manual elevator down";
END_REGION
END_FUNCTION

FUNCTION "Output_Management" : Void   // FC2, LAD
{ S7_Optimized_Access := 'TRUE' }
VERSION : 0.1
BEGIN

REGION Network 1
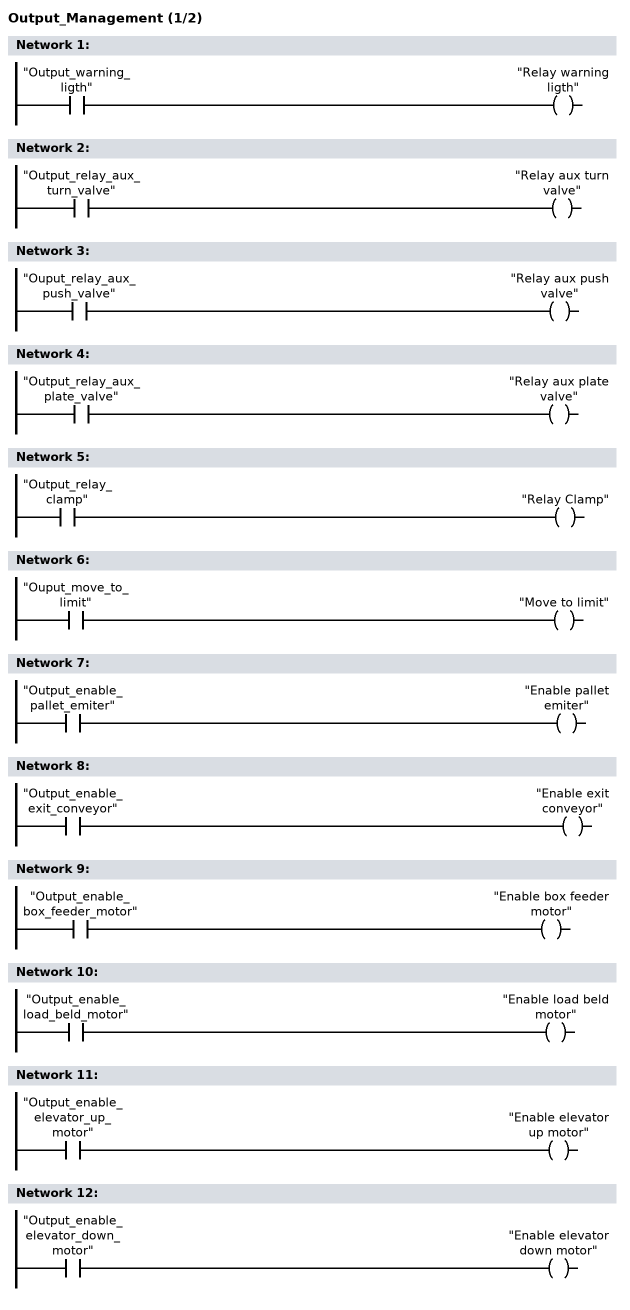
   RUNG wire#powerrail
      Contact( "Output_warning_ligth" )
      Coil( "Relay warning ligth" )
   END_RUNG
   // the same network as SCL:
   "Relay warning ligth" := "Output_warning_ligth";
END_REGION

REGION Network 2
   RUNG wire#powerrail
      Contact( "Output_relay_aux_turn_valve" )
      Coil( "Relay aux turn valve" )
   END_RUNG
   // the same network as SCL:
   "Relay aux turn valve" := "Output_relay_aux_turn_valve";
END_REGION

REGION Network 3
   RUNG wire#powerrail
      Contact( "Ouput_relay_aux_push_valve" )
      Coil( "Relay aux push valve" )
   END_RUNG
   // the same network as SCL:
   "Relay aux push valve" := "Ouput_relay_aux_push_valve";
END_REGION

REGION Network 4
   RUNG wire#powerrail
      Contact( "Output_relay_aux_plate_valve" )
      Coil( "Relay aux plate valve" )
   END_RUNG
   // the same network as SCL:
   "Relay aux plate valve" := "Output_relay_aux_plate_valve";
END_REGION

REGION Network 5
   RUNG wire#powerrail
      Contact( "Output_relay_clamp" )
      Coil( "Relay Clamp" )
   END_RUNG
   // the same network as SCL:
   "Relay Clamp" := "Output_relay_clamp";
END_REGION

REGION Network 6
   RUNG wire#powerrail
      Contact( "Ouput_move_to_limit" )
      Coil( "Move to limit" )
   END_RUNG
   // the same network as SCL:
   "Move to limit" := "Ouput_move_to_limit";
END_REGION

REGION Network 7
   RUNG wire#powerrail
      Contact( "Output_enable_pallet_emiter" )
      Coil( "Enable pallet emiter" )
   END_RUNG
   // the same network as SCL:
   "Enable pallet emiter" := "Output_enable_pallet_emiter";
END_REGION

REGION Network 8
   RUNG wire#powerrail
      Contact( "Output_enable_exit_conveyor" )
      Coil( "Enable exit conveyor" )
   END_RUNG
   // the same network as SCL:
   "Enable exit conveyor" := "Output_enable_exit_conveyor";
END_REGION

REGION Network 9
   RUNG wire#powerrail
      Contact( "Output_enable_box_feeder_motor" )
      Coil( "Enable box feeder motor" )
   END_RUNG
   // the same network as SCL:
   "Enable box feeder motor" := "Output_enable_box_feeder_motor";
END_REGION

REGION Network 10
   RUNG wire#powerrail
      Contact( "Output_enable_load_beld_motor" )
      Coil( "Enable load beld motor" )
   END_RUNG
   // the same network as SCL:
   "Enable load beld motor" := "Output_enable_load_beld_motor";
END_REGION

REGION Network 11
   RUNG wire#powerrail
      Contact( "Output_enable_elevator_up_motor" )
      Coil( "Enable elevator up motor" )
   END_RUNG
   // the same network as SCL:
   "Enable elevator up motor" := "Output_enable_elevator_up_motor";
END_REGION

REGION Network 12
   RUNG wire#powerrail
      Contact( "Output_enable_elevator_down_motor" )
      Coil( "Enable elevator down motor" )
   END_RUNG
   // the same network as SCL:
   "Enable elevator down motor" := "Output_enable_elevator_down_motor";
END_REGION

REGION Network 13
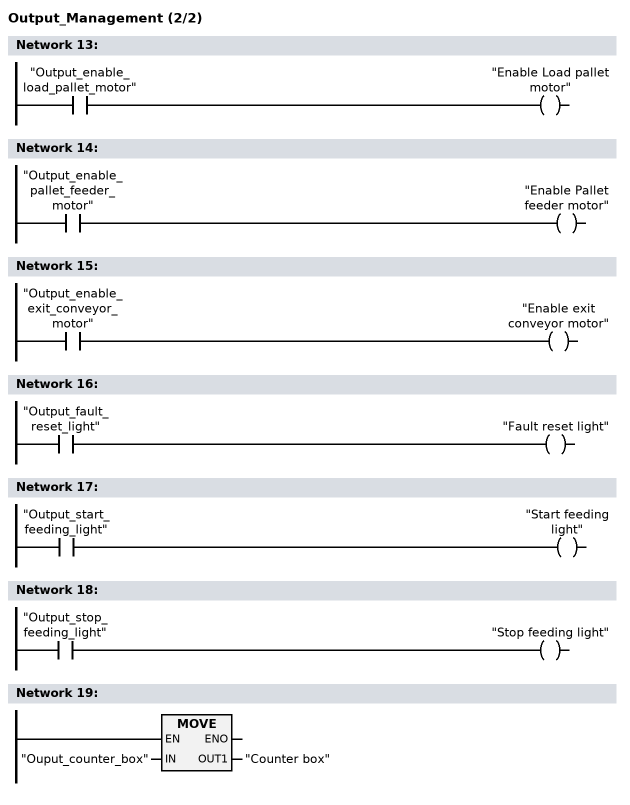
   RUNG wire#powerrail
      Contact( "Output_enable_load_pallet_motor" )
      Coil( "Enable Load pallet motor" )
   END_RUNG
   // the same network as SCL:
   "Enable Load pallet motor" := "Output_enable_load_pallet_motor";
END_REGION

REGION Network 14
   RUNG wire#powerrail
      Contact( "Output_enable_pallet_feeder_motor" )
      Coil( "Enable Pallet feeder motor" )
   END_RUNG
   // the same network as SCL:
   "Enable Pallet feeder motor" := "Output_enable_pallet_feeder_motor";
END_REGION

REGION Network 15
   RUNG wire#powerrail
      Contact( "Output_enable_exit_conveyor_motor" )
      Coil( "Enable exit conveyor motor" )
   END_RUNG
   // the same network as SCL:
   "Enable exit conveyor motor" := "Output_enable_exit_conveyor_motor";
END_REGION

REGION Network 16
   RUNG wire#powerrail
      Contact( "Output_fault_reset_light" )
      Coil( "Fault reset light" )
   END_RUNG
   // the same network as SCL:
   "Fault reset light" := "Output_fault_reset_light";
END_REGION

REGION Network 17
   RUNG wire#powerrail
      Contact( "Output_start_feeding_light" )
      Coil( "Start feeding light" )
   END_RUNG
   // the same network as SCL:
   "Start feeding light" := "Output_start_feeding_light";
END_REGION

REGION Network 18
   RUNG wire#powerrail
      Contact( "Output_stop_feeding_light" )
      Coil( "Stop feeding light" )
   END_RUNG
   // the same network as SCL:
   "Stop feeding light" := "Output_stop_feeding_light";
END_REGION

REGION Network 19
   RUNG wire#powerrail
      Move(in := "Ouput_counter_box", out1 => "Counter box")
   END_RUNG
   // the same network as SCL:
   "Counter box" := "Ouput_counter_box";
END_REGION
END_FUNCTION

FUNCTION "Module_security" : Void   // FC3, LAD
{ S7_Optimized_Access := 'TRUE' }
VERSION : 0.1
BEGIN

REGION Network 1
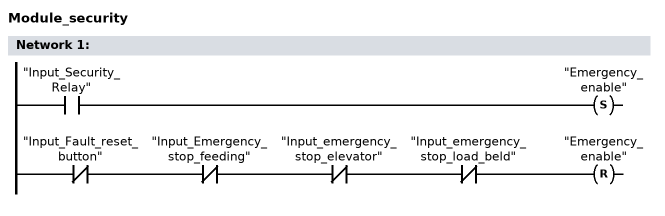
   RUNG wire#powerrail
      Contact( "Input_Security_Relay" )
      S_Coil( "Emergency_enable" )
   END_RUNG
   RUNG wire#powerrail
      I_Contact( "Input_Fault_reset_button" )
      I_Contact( "Input_Emergency_stop_feeding" )
      I_Contact( "Input_emergency_stop_elevator" )
      I_Contact( "Input_emergency_stop_load_beld" )
      R_Coil( "Emergency_enable" )
   END_RUNG
   // the same network as SCL:
   IF "Input_Security_Relay" THEN "Emergency_enable" := TRUE; END_IF;
   IF NOT "Input_Fault_reset_button" AND NOT "Input_Emergency_stop_feeding" AND NOT "Input_emergency_stop_elevator" AND NOT "Input_emergency_stop_load_beld" THEN
       "Emergency_enable" := FALSE;
   END_IF;
END_REGION
END_FUNCTION

FUNCTION "Manual_drive_module" : Void   // FC4, LAD
{ S7_Optimized_Access := 'TRUE' }
VERSION : 0.1
   VAR_TEMP   // added for the SCL form of the ladder/FBD networks
      _w1 : Bool;
   END_VAR
BEGIN

REGION Network 1
   // Manual box feeder
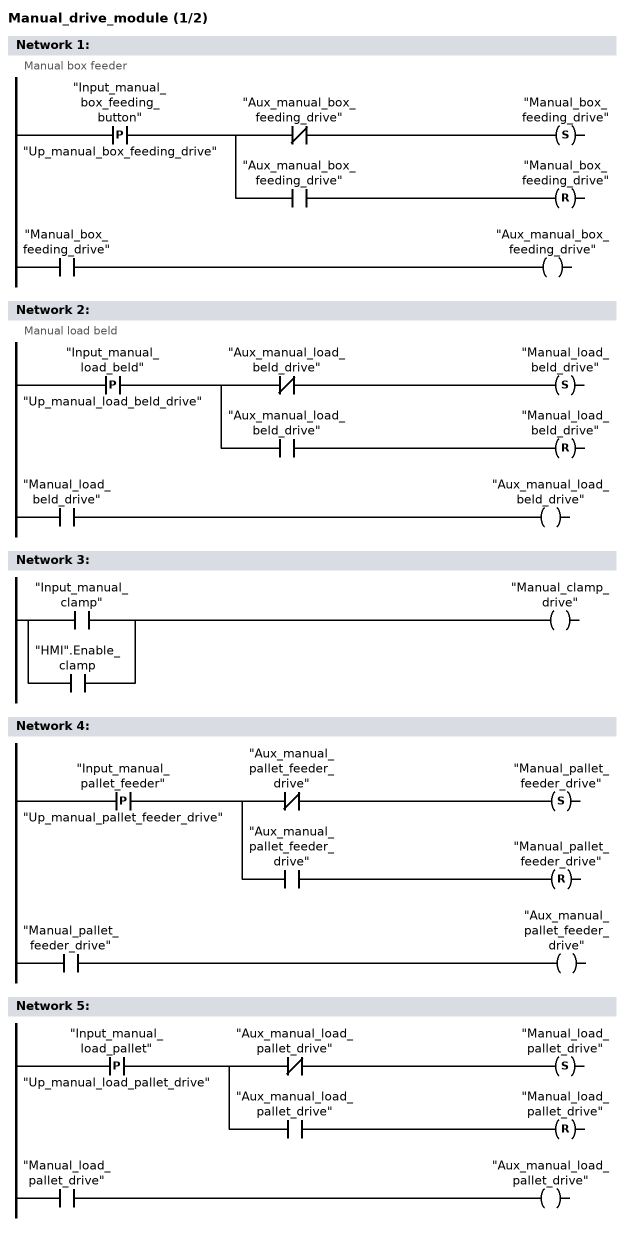
   RUNG wire#powerrail
      P_Contact(operand := "Input_manual_box_feeding_button", bit := "Up_manual_box_feeding_drive")
      wire#w1
      I_Contact( "Aux_manual_box_feeding_drive" )
      S_Coil( "Manual_box_feeding_drive" )
   END_RUNG
   RUNG wire#w1
      Contact( "Aux_manual_box_feeding_drive" )
      R_Coil( "Manual_box_feeding_drive" )
   END_RUNG
   RUNG wire#powerrail
      Contact( "Manual_box_feeding_drive" )
      Coil( "Aux_manual_box_feeding_drive" )
   END_RUNG
   // the same network as SCL:
   #_w1 := "Input_manual_box_feeding_button" AND NOT "Up_manual_box_feeding_drive";   // rising edge of "Input_manual_box_feeding_button"
   "Up_manual_box_feeding_drive" := "Input_manual_box_feeding_button";
   IF #_w1 AND NOT "Aux_manual_box_feeding_drive" THEN "Manual_box_feeding_drive" := TRUE; END_IF;
   IF #_w1 AND "Aux_manual_box_feeding_drive" THEN "Manual_box_feeding_drive" := FALSE; END_IF;
   "Aux_manual_box_feeding_drive" := "Manual_box_feeding_drive";
END_REGION

REGION Network 2
   // Manual load beld
   RUNG wire#powerrail
      P_Contact(operand := "Input_manual_load_beld", bit := "Up_manual_load_beld_drive")
      wire#w1
      I_Contact( "Aux_manual_load_beld_drive" )
      S_Coil( "Manual_load_beld_drive" )
   END_RUNG
   RUNG wire#w1
      Contact( "Aux_manual_load_beld_drive" )
      R_Coil( "Manual_load_beld_drive" )
   END_RUNG
   RUNG wire#powerrail
      Contact( "Manual_load_beld_drive" )
      Coil( "Aux_manual_load_beld_drive" )
   END_RUNG
   // the same network as SCL:
   #_w1 := "Input_manual_load_beld" AND NOT "Up_manual_load_beld_drive";   // rising edge of "Input_manual_load_beld"
   "Up_manual_load_beld_drive" := "Input_manual_load_beld";
   IF #_w1 AND NOT "Aux_manual_load_beld_drive" THEN "Manual_load_beld_drive" := TRUE; END_IF;
   IF #_w1 AND "Aux_manual_load_beld_drive" THEN "Manual_load_beld_drive" := FALSE; END_IF;
   "Aux_manual_load_beld_drive" := "Manual_load_beld_drive";
END_REGION

REGION Network 3
   RUNG wire#powerrail
      Contact( "Input_manual_clamp" )
      wire#w1
      Coil( "Manual_clamp_drive" )
   END_RUNG
   RUNG wire#powerrail
      Contact( "HMI".Enable_clamp )
   END_RUNG wire#w1
   // the same network as SCL:
   "Manual_clamp_drive" := "Input_manual_clamp" OR "HMI".Enable_clamp;
END_REGION

REGION Network 4
   RUNG wire#powerrail
      P_Contact(operand := "Input_manual_pallet_feeder", bit := "Up_manual_pallet_feeder_drive")
      wire#w1
      I_Contact( "Aux_manual_pallet_feeder_drive" )
      S_Coil( "Manual_pallet_feeder_drive" )
   END_RUNG
   RUNG wire#w1
      Contact( "Aux_manual_pallet_feeder_drive" )
      R_Coil( "Manual_pallet_feeder_drive" )
   END_RUNG
   RUNG wire#powerrail
      Contact( "Manual_pallet_feeder_drive" )
      Coil( "Aux_manual_pallet_feeder_drive" )
   END_RUNG
   // the same network as SCL:
   #_w1 := "Input_manual_pallet_feeder" AND NOT "Up_manual_pallet_feeder_drive";   // rising edge of "Input_manual_pallet_feeder"
   "Up_manual_pallet_feeder_drive" := "Input_manual_pallet_feeder";
   IF #_w1 AND NOT "Aux_manual_pallet_feeder_drive" THEN "Manual_pallet_feeder_drive" := TRUE; END_IF;
   IF #_w1 AND "Aux_manual_pallet_feeder_drive" THEN "Manual_pallet_feeder_drive" := FALSE; END_IF;
   "Aux_manual_pallet_feeder_drive" := "Manual_pallet_feeder_drive";
END_REGION

REGION Network 5
   RUNG wire#powerrail
      P_Contact(operand := "Input_manual_load_pallet", bit := "Up_manual_load_pallet_drive")
      wire#w1
      I_Contact( "Aux_manual_load_pallet_drive" )
      S_Coil( "Manual_load_pallet_drive" )
   END_RUNG
   RUNG wire#w1
      Contact( "Aux_manual_load_pallet_drive" )
      R_Coil( "Manual_load_pallet_drive" )
   END_RUNG
   RUNG wire#powerrail
      Contact( "Manual_load_pallet_drive" )
      Coil( "Aux_manual_load_pallet_drive" )
   END_RUNG
   // the same network as SCL:
   #_w1 := "Input_manual_load_pallet" AND NOT "Up_manual_load_pallet_drive";   // rising edge of "Input_manual_load_pallet"
   "Up_manual_load_pallet_drive" := "Input_manual_load_pallet";
   IF #_w1 AND NOT "Aux_manual_load_pallet_drive" THEN "Manual_load_pallet_drive" := TRUE; END_IF;
   IF #_w1 AND "Aux_manual_load_pallet_drive" THEN "Manual_load_pallet_drive" := FALSE; END_IF;
   "Aux_manual_load_pallet_drive" := "Manual_load_pallet_drive";
END_REGION

REGION Network 6
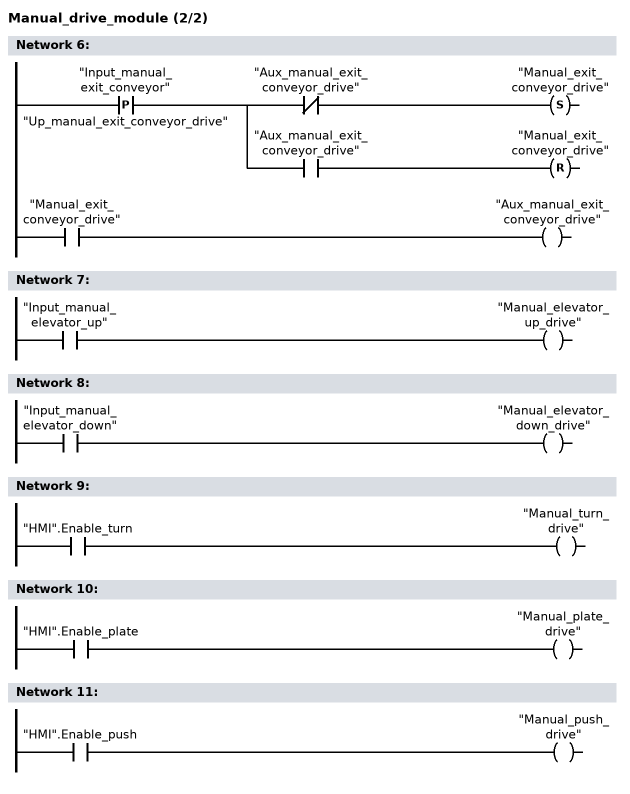
   RUNG wire#powerrail
      P_Contact(operand := "Input_manual_exit_conveyor", bit := "Up_manual_exit_conveyor_drive")
      wire#w1
      I_Contact( "Aux_manual_exit_conveyor_drive" )
      S_Coil( "Manual_exit_conveyor_drive" )
   END_RUNG
   RUNG wire#w1
      Contact( "Aux_manual_exit_conveyor_drive" )
      R_Coil( "Manual_exit_conveyor_drive" )
   END_RUNG
   RUNG wire#powerrail
      Contact( "Manual_exit_conveyor_drive" )
      Coil( "Aux_manual_exit_conveyor_drive" )
   END_RUNG
   // the same network as SCL:
   #_w1 := "Input_manual_exit_conveyor" AND NOT "Up_manual_exit_conveyor_drive";   // rising edge of "Input_manual_exit_conveyor"
   "Up_manual_exit_conveyor_drive" := "Input_manual_exit_conveyor";
   IF #_w1 AND NOT "Aux_manual_exit_conveyor_drive" THEN "Manual_exit_conveyor_drive" := TRUE; END_IF;
   IF #_w1 AND "Aux_manual_exit_conveyor_drive" THEN "Manual_exit_conveyor_drive" := FALSE; END_IF;
   "Aux_manual_exit_conveyor_drive" := "Manual_exit_conveyor_drive";
END_REGION

REGION Network 7
   RUNG wire#powerrail
      Contact( "Input_manual_elevator_up" )
      Coil( "Manual_elevator_up_drive" )
   END_RUNG
   // the same network as SCL:
   "Manual_elevator_up_drive" := "Input_manual_elevator_up";
END_REGION

REGION Network 8
   RUNG wire#powerrail
      Contact( "Input_manual_elevator_down" )
      Coil( "Manual_elevator_down_drive" )
   END_RUNG
   // the same network as SCL:
   "Manual_elevator_down_drive" := "Input_manual_elevator_down";
END_REGION

REGION Network 9
   RUNG wire#powerrail
      Contact( "HMI".Enable_turn )
      Coil( "Manual_turn_drive" )
   END_RUNG
   // the same network as SCL:
   "Manual_turn_drive" := "HMI".Enable_turn;
END_REGION

REGION Network 10
   RUNG wire#powerrail
      Contact( "HMI".Enable_plate )
      Coil( "Manual_plate_drive" )
   END_RUNG
   // the same network as SCL:
   "Manual_plate_drive" := "HMI".Enable_plate;
END_REGION

REGION Network 11
   RUNG wire#powerrail
      Contact( "HMI".Enable_push )
      Coil( "Manual_push_drive" )
   END_RUNG
   // the same network as SCL:
   "Manual_push_drive" := "HMI".Enable_push;
END_REGION
END_FUNCTION

FUNCTION "Output_drives" : Void   // FC5, LAD
{ S7_Optimized_Access := 'TRUE' }
VERSION : 0.1
BEGIN

REGION Network 1
   // Drive box feeding
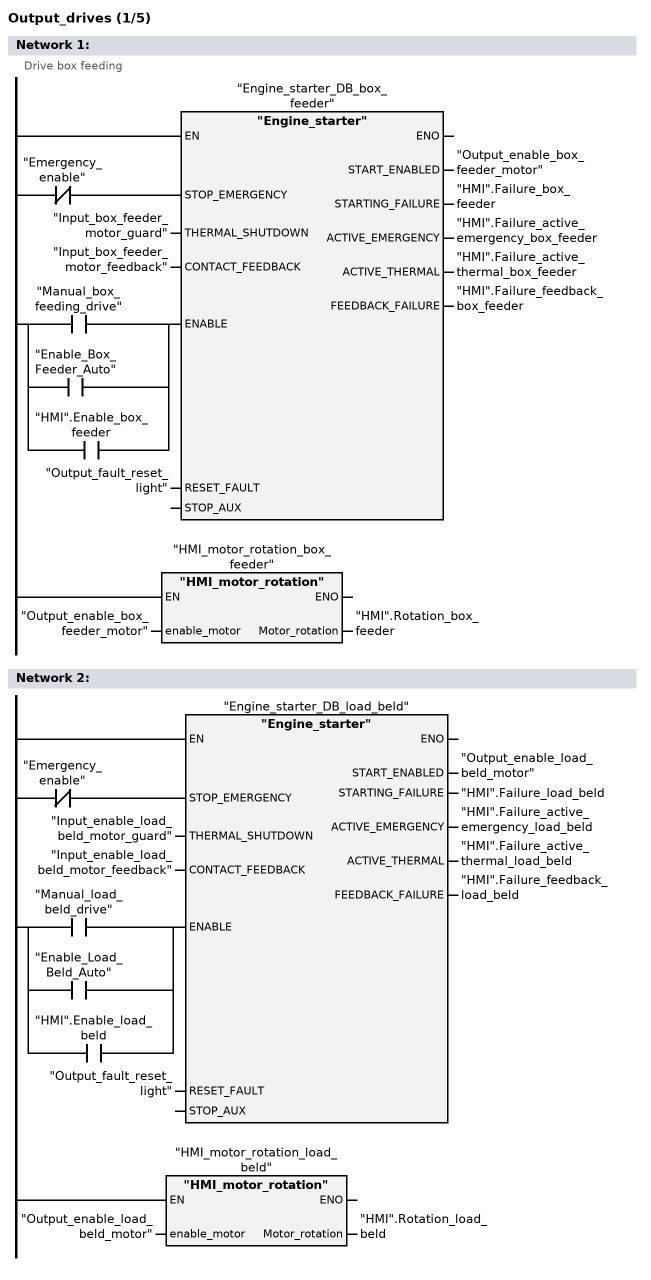
   RUNG wire#powerrail
      "Engine_starter_DB_box_feeder"(STOP_EMERGENCY := wire#w1, ENABLE := wire#w2, THERMAL_SHUTDOWN := "Input_box_feeder_motor_guard", CONTACT_FEEDBACK := "Input_box_feeder_motor_feedback", RESET_FAULT := "Output_fault_reset_light", STOP_AUX :=, START_ENABLED => "Output_enable_box_feeder_motor", STARTING_FAILURE => "HMI".Failure_box_feeder, ACTIVE_EMERGENCY => "HMI".Failure_active_emergency_box_feeder, ACTIVE_THERMAL => "HMI".Failure_active_thermal_box_feeder, FEEDBACK_FAILURE => "HMI".Failure_feedback_box_feeder)
   END_RUNG
   RUNG wire#powerrail
      I_Contact( "Emergency_enable" )
   END_RUNG wire#w1
   RUNG wire#powerrail
      Contact( "Manual_box_feeding_drive" )
   END_RUNG wire#w2
   RUNG wire#powerrail
      Contact( "Enable_Box_Feeder_Auto" )
   END_RUNG wire#w2
   RUNG wire#powerrail
      Contact( "HMI".Enable_box_feeder )
   END_RUNG wire#w2
   RUNG wire#powerrail
      "HMI_motor_rotation_box_feeder"(enable_motor := "Output_enable_box_feeder_motor", Motor_rotation => "HMI".Rotation_box_feeder)
   END_RUNG
   // the same network as SCL:
   "Engine_starter_DB_box_feeder"(STOP_EMERGENCY := NOT "Emergency_enable",   // "Engine_starter"
                           THERMAL_SHUTDOWN := "Input_box_feeder_motor_guard",
                           CONTACT_FEEDBACK := "Input_box_feeder_motor_feedback",
                           ENABLE := "Manual_box_feeding_drive" OR "Enable_Box_Feeder_Auto" OR "HMI".Enable_box_feeder,
                           RESET_FAULT := "Output_fault_reset_light",
                           START_ENABLED => "Output_enable_box_feeder_motor",
                           STARTING_FAILURE => "HMI".Failure_box_feeder,
                           ACTIVE_EMERGENCY => "HMI".Failure_active_emergency_box_feeder,
                           ACTIVE_THERMAL => "HMI".Failure_active_thermal_box_feeder,
                           FEEDBACK_FAILURE => "HMI".Failure_feedback_box_feeder);
   "HMI_motor_rotation_box_feeder"(enable_motor := "Output_enable_box_feeder_motor",   // "HMI_motor_rotation"
                           Motor_rotation => "HMI".Rotation_box_feeder);
END_REGION

REGION Network 2
   RUNG wire#powerrail
      "Engine_starter_DB_load_beld"(STOP_EMERGENCY := wire#w1, ENABLE := wire#w2, THERMAL_SHUTDOWN := "Input_enable_load_beld_motor_guard", CONTACT_FEEDBACK := "Input_enable_load_beld_motor_feedback", RESET_FAULT := "Output_fault_reset_light", STOP_AUX :=, START_ENABLED => "Output_enable_load_beld_motor", STARTING_FAILURE => "HMI".Failure_load_beld, ACTIVE_EMERGENCY => "HMI".Failure_active_emergency_load_beld, ACTIVE_THERMAL => "HMI".Failure_active_thermal_load_beld, FEEDBACK_FAILURE => "HMI".Failure_feedback_load_beld)
   END_RUNG
   RUNG wire#powerrail
      I_Contact( "Emergency_enable" )
   END_RUNG wire#w1
   RUNG wire#powerrail
      Contact( "Manual_load_beld_drive" )
   END_RUNG wire#w2
   RUNG wire#powerrail
      Contact( "Enable_Load_Beld_Auto" )
   END_RUNG wire#w2
   RUNG wire#powerrail
      Contact( "HMI".Enable_load_beld )
   END_RUNG wire#w2
   RUNG wire#powerrail
      "HMI_motor_rotation_load_beld"(enable_motor := "Output_enable_load_beld_motor", Motor_rotation => "HMI".Rotation_load_beld)
   END_RUNG
   // the same network as SCL:
   "Engine_starter_DB_load_beld"(STOP_EMERGENCY := NOT "Emergency_enable",   // "Engine_starter"
                           THERMAL_SHUTDOWN := "Input_enable_load_beld_motor_guard",
                           CONTACT_FEEDBACK := "Input_enable_load_beld_motor_feedback",
                           ENABLE := "Manual_load_beld_drive" OR "Enable_Load_Beld_Auto" OR "HMI".Enable_load_beld,
                           RESET_FAULT := "Output_fault_reset_light",
                           START_ENABLED => "Output_enable_load_beld_motor",
                           STARTING_FAILURE => "HMI".Failure_load_beld,
                           ACTIVE_EMERGENCY => "HMI".Failure_active_emergency_load_beld,
                           ACTIVE_THERMAL => "HMI".Failure_active_thermal_load_beld,
                           FEEDBACK_FAILURE => "HMI".Failure_feedback_load_beld);
   "HMI_motor_rotation_load_beld"(enable_motor := "Output_enable_load_beld_motor",   // "HMI_motor_rotation"
                           Motor_rotation => "HMI".Rotation_load_beld);
END_REGION

REGION Network 3
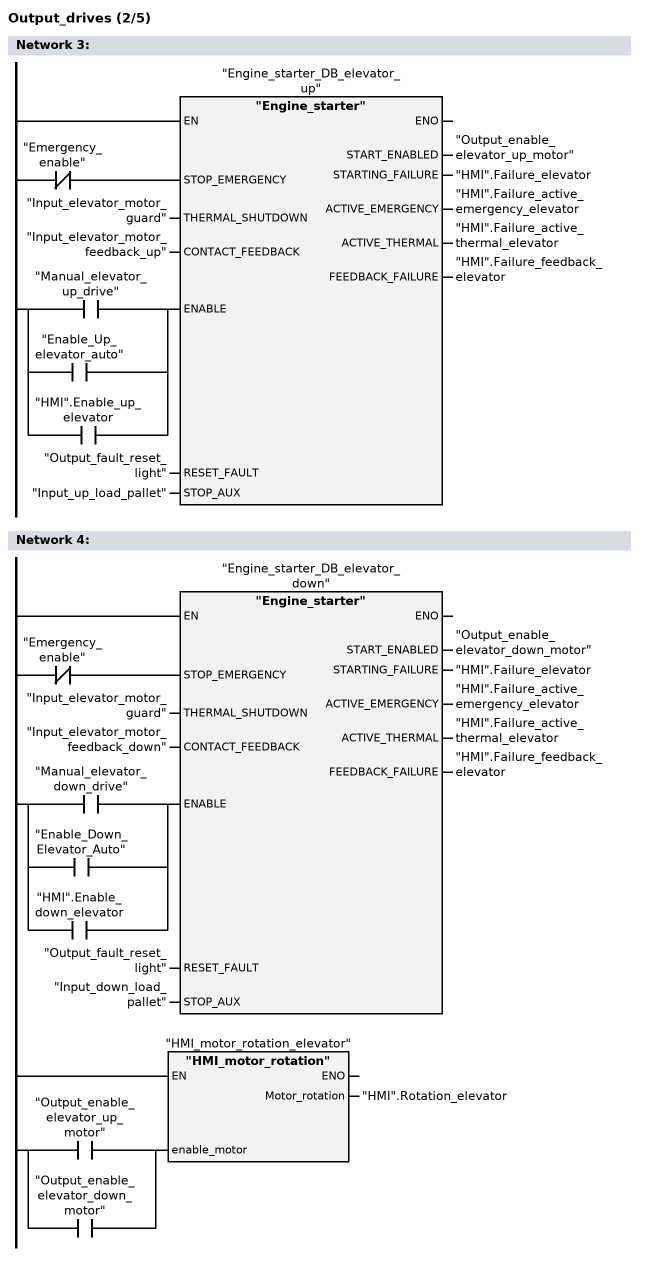
   RUNG wire#powerrail
      "Engine_starter_DB_elevator_up"(STOP_EMERGENCY := wire#w1, ENABLE := wire#w2, THERMAL_SHUTDOWN := "Input_elevator_motor_guard", CONTACT_FEEDBACK := "Input_elevator_motor_feedback_up", RESET_FAULT := "Output_fault_reset_light", STOP_AUX := "Input_up_load_pallet", START_ENABLED => "Output_enable_elevator_up_motor", STARTING_FAILURE => "HMI".Failure_elevator, ACTIVE_EMERGENCY => "HMI".Failure_active_emergency_elevator, ACTIVE_THERMAL => "HMI".Failure_active_thermal_elevator, FEEDBACK_FAILURE => "HMI".Failure_feedback_elevator)
   END_RUNG
   RUNG wire#powerrail
      I_Contact( "Emergency_enable" )
   END_RUNG wire#w1
   RUNG wire#powerrail
      Contact( "Manual_elevator_up_drive" )
   END_RUNG wire#w2
   RUNG wire#powerrail
      Contact( "Enable_Up_elevator_auto" )
   END_RUNG wire#w2
   RUNG wire#powerrail
      Contact( "HMI".Enable_up_elevator )
   END_RUNG wire#w2
   // the same network as SCL:
   "Engine_starter_DB_elevator_up"(STOP_EMERGENCY := NOT "Emergency_enable",   // "Engine_starter"
                           THERMAL_SHUTDOWN := "Input_elevator_motor_guard",
                           CONTACT_FEEDBACK := "Input_elevator_motor_feedback_up",
                           ENABLE := "Manual_elevator_up_drive" OR "Enable_Up_elevator_auto" OR "HMI".Enable_up_elevator,
                           RESET_FAULT := "Output_fault_reset_light",
                           STOP_AUX := "Input_up_load_pallet",
                           START_ENABLED => "Output_enable_elevator_up_motor",
                           STARTING_FAILURE => "HMI".Failure_elevator,
                           ACTIVE_EMERGENCY => "HMI".Failure_active_emergency_elevator,
                           ACTIVE_THERMAL => "HMI".Failure_active_thermal_elevator,
                           FEEDBACK_FAILURE => "HMI".Failure_feedback_elevator);
END_REGION

REGION Network 4
   RUNG wire#powerrail
      "Engine_starter_DB_elevator_down"(STOP_EMERGENCY := wire#w1, ENABLE := wire#w2, THERMAL_SHUTDOWN := "Input_elevator_motor_guard", CONTACT_FEEDBACK := "Input_elevator_motor_feedback_down", RESET_FAULT := "Output_fault_reset_light", STOP_AUX := "Input_down_load_pallet", START_ENABLED => "Output_enable_elevator_down_motor", STARTING_FAILURE => "HMI".Failure_elevator, ACTIVE_EMERGENCY => "HMI".Failure_active_emergency_elevator, ACTIVE_THERMAL => "HMI".Failure_active_thermal_elevator, FEEDBACK_FAILURE => "HMI".Failure_feedback_elevator)
   END_RUNG
   RUNG wire#powerrail
      I_Contact( "Emergency_enable" )
   END_RUNG wire#w1
   RUNG wire#powerrail
      Contact( "Manual_elevator_down_drive" )
   END_RUNG wire#w2
   RUNG wire#powerrail
      Contact( "Enable_Down_Elevator_Auto" )
   END_RUNG wire#w2
   RUNG wire#powerrail
      Contact( "HMI".Enable_down_elevator )
   END_RUNG wire#w2
   RUNG wire#powerrail
      "HMI_motor_rotation_elevator"(enable_motor := wire#w3, Motor_rotation => "HMI".Rotation_elevator)
   END_RUNG
   RUNG wire#powerrail
      Contact( "Output_enable_elevator_up_motor" )
   END_RUNG wire#w3
   RUNG wire#powerrail
      Contact( "Output_enable_elevator_down_motor" )
   END_RUNG wire#w3
   // the same network as SCL:
   "Engine_starter_DB_elevator_down"(STOP_EMERGENCY := NOT "Emergency_enable",   // "Engine_starter"
                           THERMAL_SHUTDOWN := "Input_elevator_motor_guard",
                           CONTACT_FEEDBACK := "Input_elevator_motor_feedback_down",
                           ENABLE := "Manual_elevator_down_drive" OR "Enable_Down_Elevator_Auto" OR "HMI".Enable_down_elevator,
                           RESET_FAULT := "Output_fault_reset_light",
                           STOP_AUX := "Input_down_load_pallet",
                           START_ENABLED => "Output_enable_elevator_down_motor",
                           STARTING_FAILURE => "HMI".Failure_elevator,
                           ACTIVE_EMERGENCY => "HMI".Failure_active_emergency_elevator,
                           ACTIVE_THERMAL => "HMI".Failure_active_thermal_elevator,
                           FEEDBACK_FAILURE => "HMI".Failure_feedback_elevator);
   "HMI_motor_rotation_elevator"(enable_motor := "Output_enable_elevator_up_motor" OR "Output_enable_elevator_down_motor",   // "HMI_motor_rotation"
                           Motor_rotation => "HMI".Rotation_elevator);
END_REGION

REGION Network 5
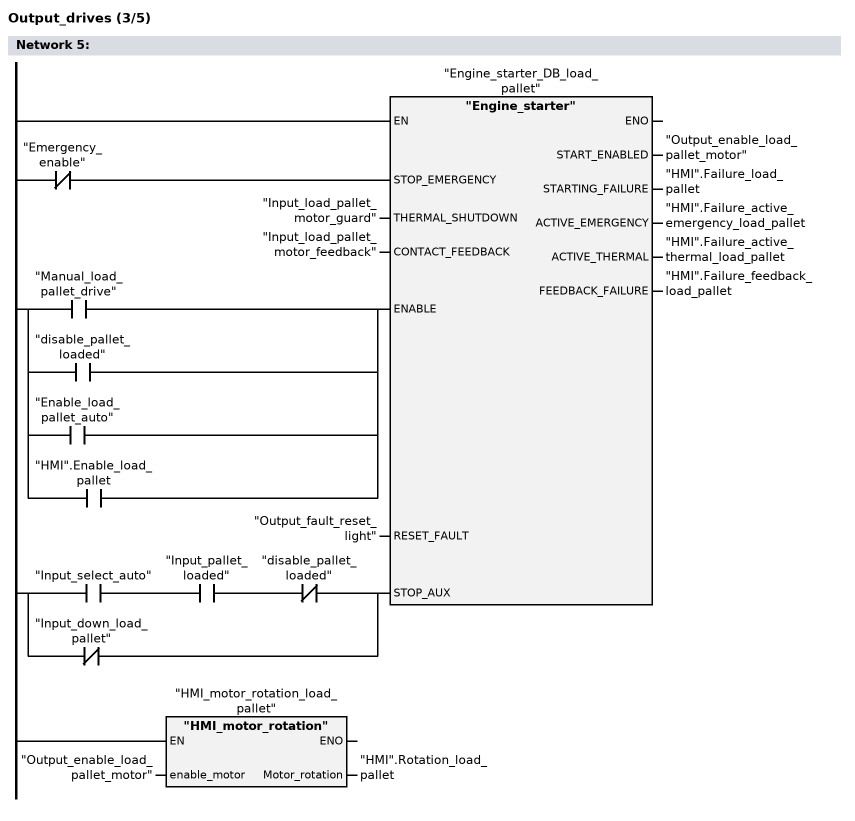
   RUNG wire#powerrail
      "Engine_starter_DB_load_pallet"(STOP_EMERGENCY := wire#w1, ENABLE := wire#w2, STOP_AUX := wire#w3, THERMAL_SHUTDOWN := "Input_load_pallet_motor_guard", CONTACT_FEEDBACK := "Input_load_pallet_motor_feedback", RESET_FAULT := "Output_fault_reset_light", START_ENABLED => "Output_enable_load_pallet_motor", STARTING_FAILURE => "HMI".Failure_load_pallet, ACTIVE_EMERGENCY => "HMI".Failure_active_emergency_load_pallet, ACTIVE_THERMAL => "HMI".Failure_active_thermal_load_pallet, FEEDBACK_FAILURE => "HMI".Failure_feedback_load_pallet)
   END_RUNG
   RUNG wire#powerrail
      I_Contact( "Emergency_enable" )
   END_RUNG wire#w1
   RUNG wire#powerrail
      Contact( "Manual_load_pallet_drive" )
   END_RUNG wire#w2
   RUNG wire#powerrail
      Contact( "disable_pallet_loaded" )
   END_RUNG wire#w2
   RUNG wire#powerrail
      Contact( "Enable_load_pallet_auto" )
   END_RUNG wire#w2
   RUNG wire#powerrail
      Contact( "HMI".Enable_load_pallet )
   END_RUNG wire#w2
   RUNG wire#powerrail
      Contact( "Input_select_auto" )
      Contact( "Input_pallet_loaded" )
      I_Contact( "disable_pallet_loaded" )
   END_RUNG wire#w3
   RUNG wire#powerrail
      I_Contact( "Input_down_load_pallet" )
   END_RUNG wire#w3
   RUNG wire#powerrail
      "HMI_motor_rotation_load_pallet"(enable_motor := "Output_enable_load_pallet_motor", Motor_rotation => "HMI".Rotation_load_pallet)
   END_RUNG
   // the same network as SCL:
   "Engine_starter_DB_load_pallet"(STOP_EMERGENCY := NOT "Emergency_enable",   // "Engine_starter"
                           THERMAL_SHUTDOWN := "Input_load_pallet_motor_guard",
                           CONTACT_FEEDBACK := "Input_load_pallet_motor_feedback",
                           ENABLE := "Manual_load_pallet_drive" OR "disable_pallet_loaded" OR "Enable_load_pallet_auto" OR "HMI".Enable_load_pallet,
                           RESET_FAULT := "Output_fault_reset_light",
                           STOP_AUX := ("Input_select_auto" AND "Input_pallet_loaded" AND NOT "disable_pallet_loaded") OR NOT "Input_down_load_pallet",
                           START_ENABLED => "Output_enable_load_pallet_motor",
                           STARTING_FAILURE => "HMI".Failure_load_pallet,
                           ACTIVE_EMERGENCY => "HMI".Failure_active_emergency_load_pallet,
                           ACTIVE_THERMAL => "HMI".Failure_active_thermal_load_pallet,
                           FEEDBACK_FAILURE => "HMI".Failure_feedback_load_pallet);
   "HMI_motor_rotation_load_pallet"(enable_motor := "Output_enable_load_pallet_motor",   // "HMI_motor_rotation"
                           Motor_rotation => "HMI".Rotation_load_pallet);
END_REGION

REGION Network 6
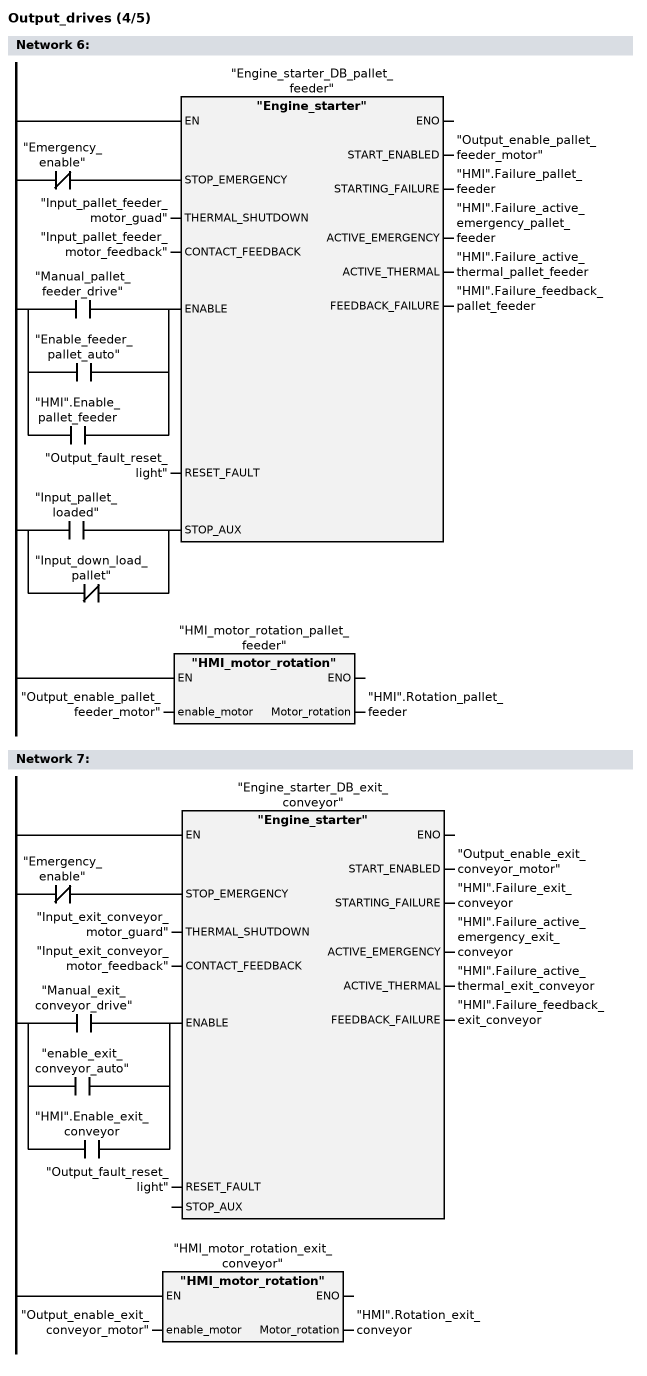
   RUNG wire#powerrail
      "Engine_starter_DB_pallet_feeder"(STOP_EMERGENCY := wire#w1, ENABLE := wire#w2, STOP_AUX := wire#w3, THERMAL_SHUTDOWN := "Input_pallet_feeder_motor_guad", CONTACT_FEEDBACK := "Input_pallet_feeder_motor_feedback", RESET_FAULT := "Output_fault_reset_light", START_ENABLED => "Output_enable_pallet_feeder_motor", STARTING_FAILURE => "HMI".Failure_pallet_feeder, ACTIVE_EMERGENCY => "HMI".Failure_active_emergency_pallet_feeder, ACTIVE_THERMAL => "HMI".Failure_active_thermal_pallet_feeder, FEEDBACK_FAILURE => "HMI".Failure_feedback_pallet_feeder)
   END_RUNG
   RUNG wire#powerrail
      I_Contact( "Emergency_enable" )
   END_RUNG wire#w1
   RUNG wire#powerrail
      Contact( "Manual_pallet_feeder_drive" )
   END_RUNG wire#w2
   RUNG wire#powerrail
      Contact( "Enable_feeder_pallet_auto" )
   END_RUNG wire#w2
   RUNG wire#powerrail
      Contact( "HMI".Enable_pallet_feeder )
   END_RUNG wire#w2
   RUNG wire#powerrail
      Contact( "Input_pallet_loaded" )
   END_RUNG wire#w3
   RUNG wire#powerrail
      I_Contact( "Input_down_load_pallet" )
   END_RUNG wire#w3
   RUNG wire#powerrail
      "HMI_motor_rotation_pallet_feeder"(enable_motor := "Output_enable_pallet_feeder_motor", Motor_rotation => "HMI".Rotation_pallet_feeder)
   END_RUNG
   // the same network as SCL:
   "Engine_starter_DB_pallet_feeder"(STOP_EMERGENCY := NOT "Emergency_enable",   // "Engine_starter"
                           THERMAL_SHUTDOWN := "Input_pallet_feeder_motor_guad",
                           CONTACT_FEEDBACK := "Input_pallet_feeder_motor_feedback",
                           ENABLE := "Manual_pallet_feeder_drive" OR "Enable_feeder_pallet_auto" OR "HMI".Enable_pallet_feeder,
                           RESET_FAULT := "Output_fault_reset_light",
                           STOP_AUX := "Input_pallet_loaded" OR NOT "Input_down_load_pallet",
                           START_ENABLED => "Output_enable_pallet_feeder_motor",
                           STARTING_FAILURE => "HMI".Failure_pallet_feeder,
                           ACTIVE_EMERGENCY => "HMI".Failure_active_emergency_pallet_feeder,
                           ACTIVE_THERMAL => "HMI".Failure_active_thermal_pallet_feeder,
                           FEEDBACK_FAILURE => "HMI".Failure_feedback_pallet_feeder);
   "HMI_motor_rotation_pallet_feeder"(enable_motor := "Output_enable_pallet_feeder_motor",   // "HMI_motor_rotation"
                           Motor_rotation => "HMI".Rotation_pallet_feeder);
END_REGION

REGION Network 7
   RUNG wire#powerrail
      "Engine_starter_DB_exit_conveyor"(STOP_EMERGENCY := wire#w1, ENABLE := wire#w2, THERMAL_SHUTDOWN := "Input_exit_conveyor_motor_guard", CONTACT_FEEDBACK := "Input_exit_conveyor_motor_feedback", RESET_FAULT := "Output_fault_reset_light", STOP_AUX :=, START_ENABLED => "Output_enable_exit_conveyor_motor", STARTING_FAILURE => "HMI".Failure_exit_conveyor, ACTIVE_EMERGENCY => "HMI".Failure_active_emergency_exit_conveyor, ACTIVE_THERMAL => "HMI".Failure_active_thermal_exit_conveyor, FEEDBACK_FAILURE => "HMI".Failure_feedback_exit_conveyor)
   END_RUNG
   RUNG wire#powerrail
      I_Contact( "Emergency_enable" )
   END_RUNG wire#w1
   RUNG wire#powerrail
      Contact( "Manual_exit_conveyor_drive" )
   END_RUNG wire#w2
   RUNG wire#powerrail
      Contact( "enable_exit_conveyor_auto" )
   END_RUNG wire#w2
   RUNG wire#powerrail
      Contact( "HMI".Enable_exit_conveyor )
   END_RUNG wire#w2
   RUNG wire#powerrail
      "HMI_motor_rotation_exit_conveyor"(enable_motor := "Output_enable_exit_conveyor_motor", Motor_rotation => "HMI".Rotation_exit_conveyor)
   END_RUNG
   // the same network as SCL:
   "Engine_starter_DB_exit_conveyor"(STOP_EMERGENCY := NOT "Emergency_enable",   // "Engine_starter"
                           THERMAL_SHUTDOWN := "Input_exit_conveyor_motor_guard",
                           CONTACT_FEEDBACK := "Input_exit_conveyor_motor_feedback",
                           ENABLE := "Manual_exit_conveyor_drive" OR "enable_exit_conveyor_auto" OR "HMI".Enable_exit_conveyor,
                           RESET_FAULT := "Output_fault_reset_light",
                           START_ENABLED => "Output_enable_exit_conveyor_motor",
                           STARTING_FAILURE => "HMI".Failure_exit_conveyor,
                           ACTIVE_EMERGENCY => "HMI".Failure_active_emergency_exit_conveyor,
                           ACTIVE_THERMAL => "HMI".Failure_active_thermal_exit_conveyor,
                           FEEDBACK_FAILURE => "HMI".Failure_feedback_exit_conveyor);
   "HMI_motor_rotation_exit_conveyor"(enable_motor := "Output_enable_exit_conveyor_motor",   // "HMI_motor_rotation"
                           Motor_rotation => "HMI".Rotation_exit_conveyor);
END_REGION

REGION Network 8
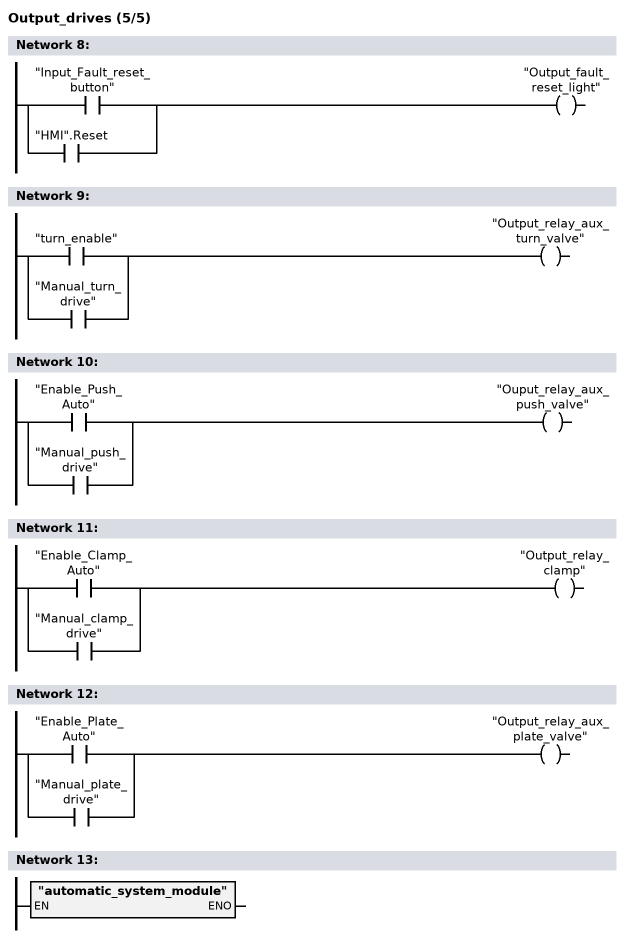
   RUNG wire#powerrail
      Contact( "Input_Fault_reset_button" )
      wire#w1
      Coil( "Output_fault_reset_light" )
   END_RUNG
   RUNG wire#powerrail
      Contact( "HMI".Reset )
   END_RUNG wire#w1
   // the same network as SCL:
   "Output_fault_reset_light" := "Input_Fault_reset_button" OR "HMI".Reset;
END_REGION

REGION Network 9
   RUNG wire#powerrail
      Contact( "turn_enable" )
      wire#w1
      Coil( "Output_relay_aux_turn_valve" )
   END_RUNG
   RUNG wire#powerrail
      Contact( "Manual_turn_drive" )
   END_RUNG wire#w1
   // the same network as SCL:
   "Output_relay_aux_turn_valve" := "turn_enable" OR "Manual_turn_drive";
END_REGION

REGION Network 10
   RUNG wire#powerrail
      Contact( "Enable_Push_Auto" )
      wire#w1
      Coil( "Ouput_relay_aux_push_valve" )
   END_RUNG
   RUNG wire#powerrail
      Contact( "Manual_push_drive" )
   END_RUNG wire#w1
   // the same network as SCL:
   "Ouput_relay_aux_push_valve" := "Enable_Push_Auto" OR "Manual_push_drive";
END_REGION

REGION Network 11
   RUNG wire#powerrail
      Contact( "Enable_Clamp_Auto" )
      wire#w1
      Coil( "Output_relay_clamp" )
   END_RUNG
   RUNG wire#powerrail
      Contact( "Manual_clamp_drive" )
   END_RUNG wire#w1
   // the same network as SCL:
   "Output_relay_clamp" := "Enable_Clamp_Auto" OR "Manual_clamp_drive";
END_REGION

REGION Network 12
   RUNG wire#powerrail
      Contact( "Enable_Plate_Auto" )
      wire#w1
      Coil( "Output_relay_aux_plate_valve" )
   END_RUNG
   RUNG wire#powerrail
      Contact( "Manual_plate_drive" )
   END_RUNG wire#w1
   // the same network as SCL:
   "Output_relay_aux_plate_valve" := "Enable_Plate_Auto" OR "Manual_plate_drive";
END_REGION

REGION Network 13
   RUNG wire#powerrail
      "automatic_system_module"()
   END_RUNG
   // the same network as SCL:
   "automatic_system_module"();
END_REGION
END_FUNCTION

FUNCTION "automatic_system_module" : Void   // FC6, LAD
{ S7_Optimized_Access := 'TRUE' }
VERSION : 0.1
   VAR_TEMP   // added for the SCL form of the ladder/FBD networks
      _w1 : Bool;
      _w2 : Bool;
      _w3 : Bool;
   END_VAR
BEGIN

REGION Network 1
   // Set zero point
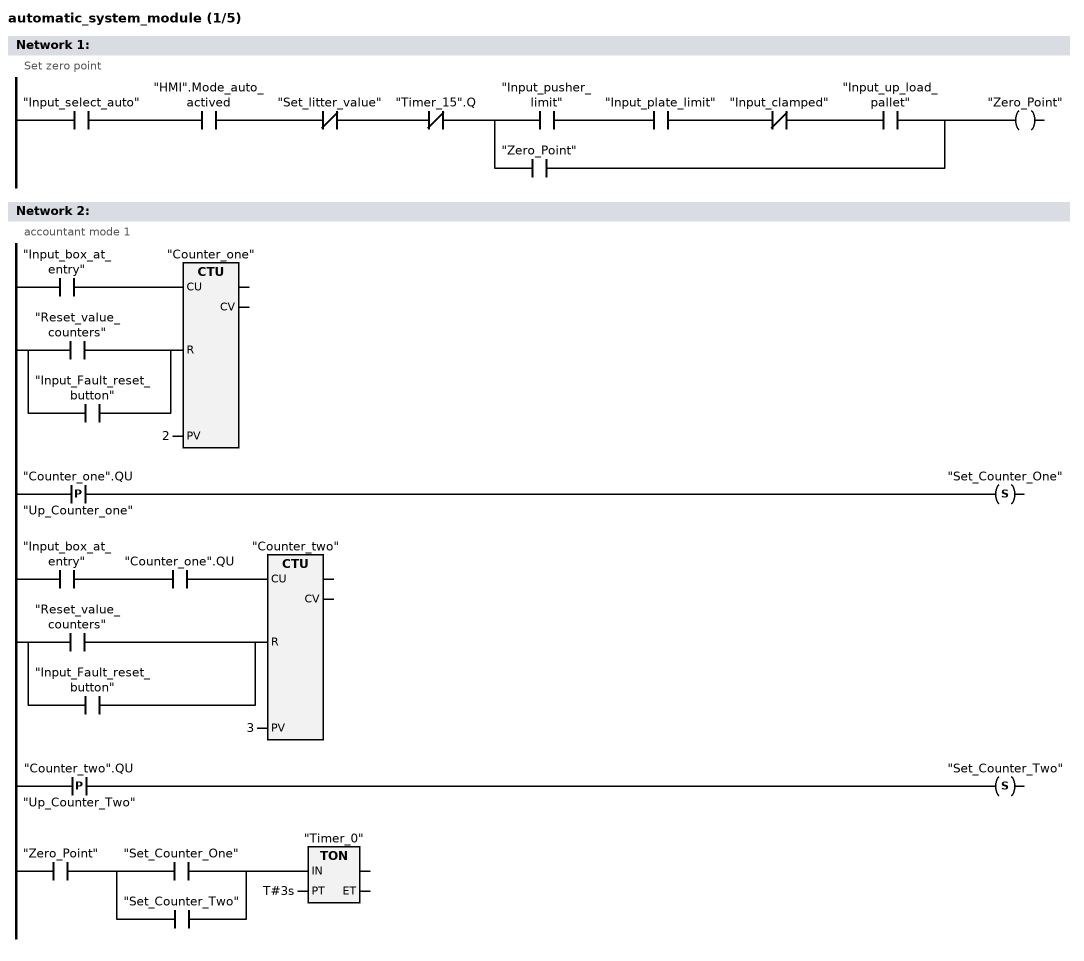
   RUNG wire#powerrail
      Contact( "Input_select_auto" )
      Contact( "HMI".Mode_auto_actived )
      I_Contact( "Set_litter_value" )
      I_Contact( "Timer_15".Q )
      wire#w1
      Contact( "Input_pusher_limit" )
      Contact( "Input_plate_limit" )
      I_Contact( "Input_clamped" )
      Contact( "Input_up_load_pallet" )
      wire#w2
      Coil( "Zero_Point" )
   END_RUNG
   RUNG wire#w1
      Contact( "Zero_Point" )
   END_RUNG wire#w2
   // the same network as SCL:
   "Zero_Point" := "Input_select_auto" AND "HMI".Mode_auto_actived AND NOT "Set_litter_value" AND NOT "Timer_15".Q AND (("Input_pusher_limit" AND "Input_plate_limit" AND NOT "Input_clamped" AND "Input_up_load_pallet") OR "Zero_Point");
END_REGION

REGION Network 2
   // accountant mode 1
   "Counter_one".CTU(CU := "Input_box_at_entry",
                     R := "Reset_value_counters" OR "Input_Fault_reset_button",
                     PV := 2);
   #_w1 := "Counter_one".QU AND NOT "Up_Counter_one";   // rising edge of "Counter_one".QU
   "Up_Counter_one" := "Counter_one".QU;
   IF #_w1 THEN "Set_Counter_One" := TRUE; END_IF;
   "Counter_two".CTU(CU := "Input_box_at_entry" AND "Counter_one".QU,
                     R := "Reset_value_counters" OR "Input_Fault_reset_button",
                     PV := 3);
   #_w2 := "Counter_two".QU AND NOT "Up_Counter_Two";   // rising edge of "Counter_two".QU
   "Up_Counter_Two" := "Counter_two".QU;
   IF #_w2 THEN "Set_Counter_Two" := TRUE; END_IF;
   "Timer_0".TON(IN := "Zero_Point" AND ("Set_Counter_One" OR "Set_Counter_Two"), PT := T#3s);
END_REGION

REGION Network 3
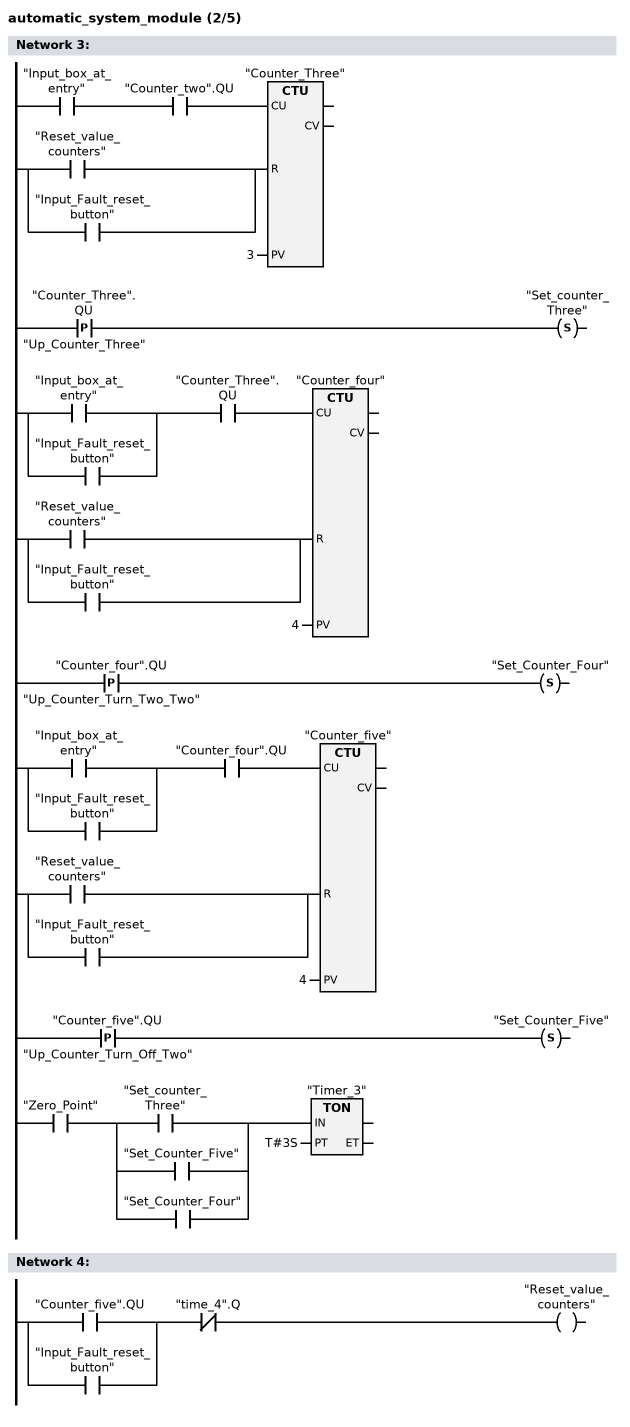
   "Counter_Three".CTU(CU := "Input_box_at_entry" AND "Counter_two".QU,
                       R := "Reset_value_counters" OR "Input_Fault_reset_button",
                       PV := 3);
   #_w1 := "Counter_Three".QU AND NOT "Up_Counter_Three";   // rising edge of "Counter_Three".QU
   "Up_Counter_Three" := "Counter_Three".QU;
   IF #_w1 THEN "Set_counter_Three" := TRUE; END_IF;
   "Counter_four".CTU(CU := ("Input_box_at_entry" OR "Input_Fault_reset_button") AND "Counter_Three".QU,
                      R := "Reset_value_counters" OR "Input_Fault_reset_button",
                      PV := 4);
   #_w2 := "Counter_four".QU AND NOT "Up_Counter_Turn_Two_Two";   // rising edge of "Counter_four".QU
   "Up_Counter_Turn_Two_Two" := "Counter_four".QU;
   IF #_w2 THEN "Set_Counter_Four" := TRUE; END_IF;
   "Counter_five".CTU(CU := ("Input_box_at_entry" OR "Input_Fault_reset_button") AND "Counter_four".QU,
                      R := "Reset_value_counters" OR "Input_Fault_reset_button",
                      PV := 4);
   #_w3 := "Counter_five".QU AND NOT "Up_Counter_Turn_Off_Two";   // rising edge of "Counter_five".QU
   "Up_Counter_Turn_Off_Two" := "Counter_five".QU;
   IF #_w3 THEN "Set_Counter_Five" := TRUE; END_IF;
   "Timer_3".TON(IN := "Zero_Point" AND ("Set_counter_Three" OR "Set_Counter_Five" OR "Set_Counter_Four"),
                 PT := T#3S);
END_REGION

REGION Network 4
   RUNG wire#powerrail
      Contact( "Counter_five".QU )
      wire#w1
      I_Contact( "time_4".Q )
      Coil( "Reset_value_counters" )
   END_RUNG
   RUNG wire#powerrail
      Contact( "Input_Fault_reset_button" )
   END_RUNG wire#w1
   // the same network as SCL:
   "Reset_value_counters" := ("Counter_five".QU OR "Input_Fault_reset_button") AND NOT "time_4".Q;
END_REGION

REGION Network 5
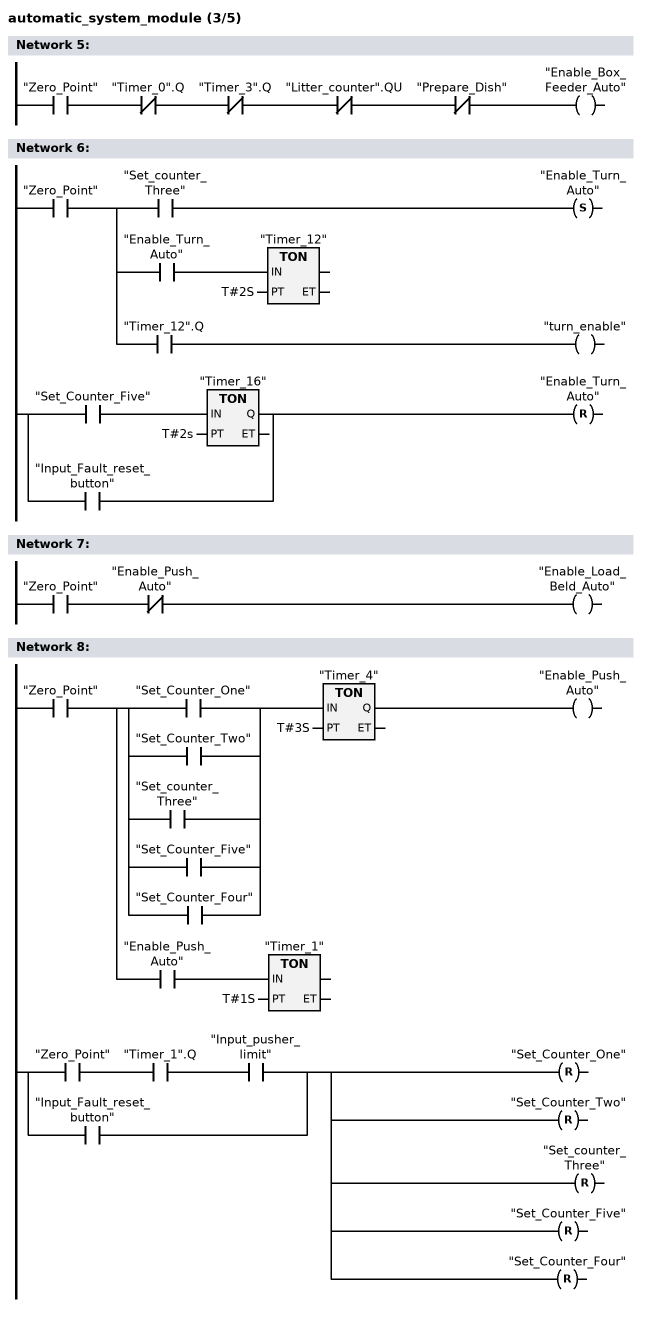
   RUNG wire#powerrail
      Contact( "Zero_Point" )
      I_Contact( "Timer_0".Q )
      I_Contact( "Timer_3".Q )
      I_Contact( "Litter_counter".QU )
      I_Contact( "Prepare_Dish" )
      Coil( "Enable_Box_Feeder_Auto" )
   END_RUNG
   // the same network as SCL:
   "Enable_Box_Feeder_Auto" := "Zero_Point" AND NOT "Timer_0".Q AND NOT "Timer_3".Q AND NOT "Litter_counter".QU AND NOT "Prepare_Dish";
END_REGION

REGION Network 6
   IF "Zero_Point" AND "Set_counter_Three" THEN "Enable_Turn_Auto" := TRUE; END_IF;
   "Timer_12".TON(IN := "Zero_Point" AND "Enable_Turn_Auto", PT := T#2S);
   "turn_enable" := "Zero_Point" AND "Timer_12".Q;
   "Timer_16".TON(IN := "Set_Counter_Five", PT := T#2s);
   IF "Timer_16".Q OR "Input_Fault_reset_button" THEN "Enable_Turn_Auto" := FALSE; END_IF;
END_REGION

REGION Network 7
   RUNG wire#powerrail
      Contact( "Zero_Point" )
      I_Contact( "Enable_Push_Auto" )
      Coil( "Enable_Load_Beld_Auto" )
   END_RUNG
   // the same network as SCL:
   "Enable_Load_Beld_Auto" := "Zero_Point" AND NOT "Enable_Push_Auto";
END_REGION

REGION Network 8
   "Timer_4".TON(IN := "Zero_Point" AND ("Set_Counter_One" OR "Set_Counter_Two" OR "Set_counter_Three" OR "Set_Counter_Five" OR "Set_Counter_Four"),
                 PT := T#3S);
   "Enable_Push_Auto" := "Timer_4".Q;
   "Timer_1".TON(IN := "Zero_Point" AND "Enable_Push_Auto", PT := T#1S);
   IF ("Zero_Point" AND "Timer_1".Q AND "Input_pusher_limit") OR "Input_Fault_reset_button" THEN
       "Set_Counter_One" := FALSE;
       "Set_Counter_Two" := FALSE;
       "Set_counter_Three" := FALSE;
       "Set_Counter_Five" := FALSE;
       "Set_Counter_Four" := FALSE;
   END_IF;
END_REGION

REGION Network 9
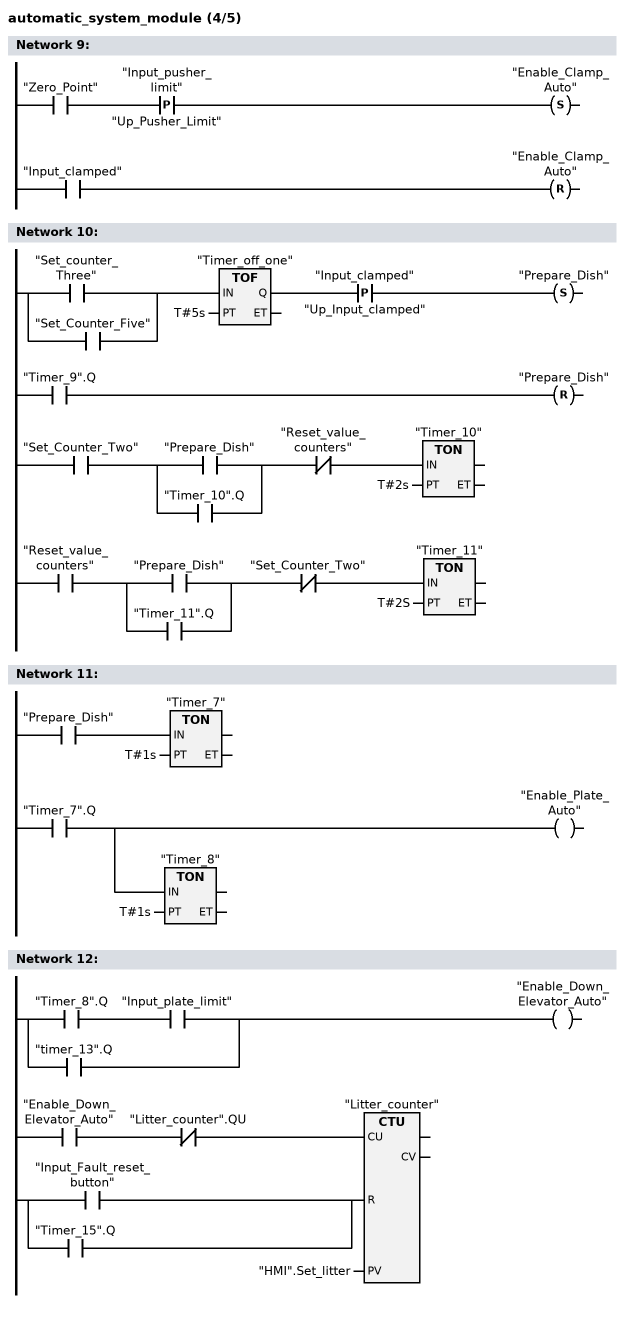
   RUNG wire#powerrail
      Contact( "Zero_Point" )
      P_Contact(operand := "Input_pusher_limit", bit := "Up_Pusher_Limit")
      S_Coil( "Enable_Clamp_Auto" )
   END_RUNG
   RUNG wire#powerrail
      Contact( "Input_clamped" )
      R_Coil( "Enable_Clamp_Auto" )
   END_RUNG
   // the same network as SCL:
   #_w1 := "Zero_Point" AND "Input_pusher_limit" AND NOT "Up_Pusher_Limit";   // rising edge of "Input_pusher_limit"
   "Up_Pusher_Limit" := "Input_pusher_limit";
   IF #_w1 THEN "Enable_Clamp_Auto" := TRUE; END_IF;
   IF "Input_clamped" THEN "Enable_Clamp_Auto" := FALSE; END_IF;
END_REGION

REGION Network 10
   "Timer_off_one".TOF(IN := "Set_counter_Three" OR "Set_Counter_Five", PT := T#5s);
   #_w1 := "Timer_off_one".Q AND "Input_clamped" AND NOT "Up_Input_clamped";   // rising edge of "Input_clamped"
   "Up_Input_clamped" := "Input_clamped";
   IF #_w1 THEN "Prepare_Dish" := TRUE; END_IF;
   IF "Timer_9".Q THEN "Prepare_Dish" := FALSE; END_IF;
   "Timer_10".TON(IN := "Set_Counter_Two" AND ("Prepare_Dish" OR "Timer_10".Q) AND NOT "Reset_value_counters",
                  PT := T#2s);
   "Timer_11".TON(IN := "Reset_value_counters" AND ("Prepare_Dish" OR "Timer_11".Q) AND NOT "Set_Counter_Two",
                  PT := T#2S);
END_REGION

REGION Network 11
   "Timer_7".TON(IN := "Prepare_Dish", PT := T#1s);
   "Enable_Plate_Auto" := "Timer_7".Q;
   "Timer_8".TON(IN := "Timer_7".Q, PT := T#1s);
END_REGION

REGION Network 12
   "Enable_Down_Elevator_Auto" := ("Timer_8".Q AND "Input_plate_limit") OR "timer_13".Q;
   "Litter_counter".CTU(CU := "Enable_Down_Elevator_Auto" AND NOT "Litter_counter".QU,
                        R := "Input_Fault_reset_button" OR "Timer_15".Q,
                        PV := "HMI".Set_litter);
END_REGION

REGION Network 13
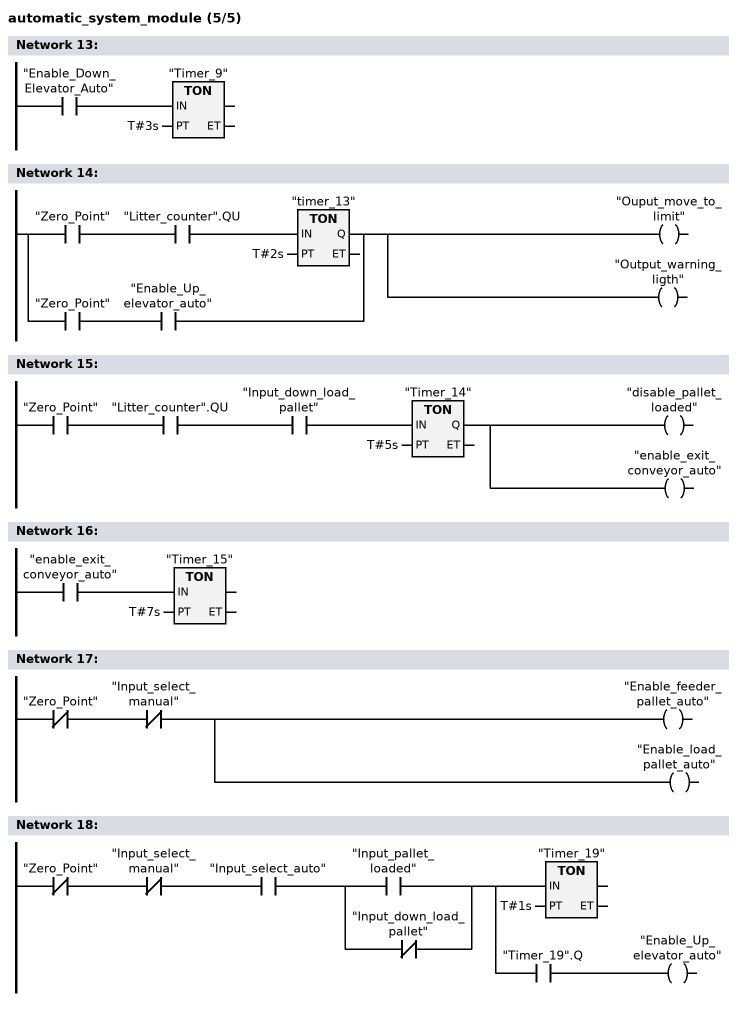
   "Timer_9".TON(IN := "Enable_Down_Elevator_Auto", PT := T#3s);
END_REGION

REGION Network 14
   "timer_13".TON(IN := "Zero_Point" AND "Litter_counter".QU, PT := T#2s);
   "Ouput_move_to_limit" := "timer_13".Q OR ("Zero_Point" AND "Enable_Up_elevator_auto");
   "Output_warning_ligth" := "Ouput_move_to_limit";
END_REGION

REGION Network 15
   "Timer_14".TON(IN := "Zero_Point" AND "Litter_counter".QU AND "Input_down_load_pallet", PT := T#5s);
   "disable_pallet_loaded" := "Timer_14".Q;
   "enable_exit_conveyor_auto" := "Timer_14".Q;
END_REGION

REGION Network 16
   "Timer_15".TON(IN := "enable_exit_conveyor_auto", PT := T#7s);
END_REGION

REGION Network 17
   RUNG wire#powerrail
      I_Contact( "Zero_Point" )
      I_Contact( "Input_select_manual" )
      wire#w1
      Coil( "Enable_feeder_pallet_auto" )
   END_RUNG
   RUNG wire#w1
      Coil( "Enable_load_pallet_auto" )
   END_RUNG
   // the same network as SCL:
   "Enable_feeder_pallet_auto" := NOT "Zero_Point" AND NOT "Input_select_manual";
   "Enable_load_pallet_auto" := "Enable_feeder_pallet_auto";
END_REGION

REGION Network 18
   #_w1 := NOT "Zero_Point" AND NOT "Input_select_manual" AND "Input_select_auto" AND ("Input_pallet_loaded" OR NOT "Input_down_load_pallet");
   "Timer_19".TON(IN := #_w1, PT := T#1s);
   "Enable_Up_elevator_auto" := #_w1 AND "Timer_19".Q;
END_REGION
END_FUNCTION

FUNCTION "Command_hmi" : Void   // FC7, LAD
{ S7_Optimized_Access := 'TRUE' }
VERSION : 0.1
   VAR_TEMP   // added for the SCL form of the ladder/FBD networks
      _w1 : Bool;
      _w2 : Bool;
      _w3 : Bool;
      _w4 : Bool;
   END_VAR
BEGIN

REGION Network 1
   // System mode manual
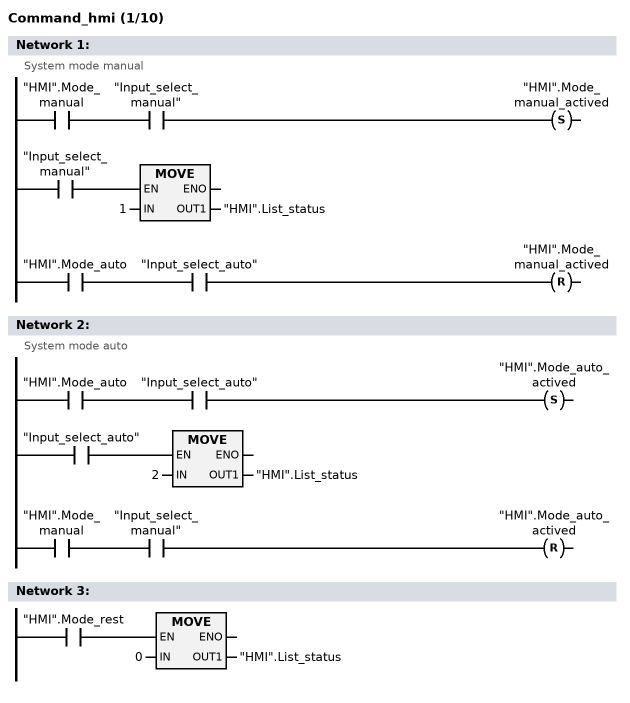
   RUNG wire#powerrail
      Contact( "HMI".Mode_manual )
      Contact( "Input_select_manual" )
      S_Coil( "HMI".Mode_manual_actived )
   END_RUNG
   RUNG wire#powerrail
      Contact( "Input_select_manual" )
      Move(in := 1, out1 => "HMI".List_status)
   END_RUNG
   RUNG wire#powerrail
      Contact( "HMI".Mode_auto )
      Contact( "Input_select_auto" )
      R_Coil( "HMI".Mode_manual_actived )
   END_RUNG
   // the same network as SCL:
   IF "HMI".Mode_manual AND "Input_select_manual" THEN "HMI".Mode_manual_actived := TRUE; END_IF;
   IF "Input_select_manual" THEN "HMI".List_status := 1; END_IF;
   IF "HMI".Mode_auto AND "Input_select_auto" THEN "HMI".Mode_manual_actived := FALSE; END_IF;
END_REGION

REGION Network 2
   // System mode auto
   RUNG wire#powerrail
      Contact( "HMI".Mode_auto )
      Contact( "Input_select_auto" )
      S_Coil( "HMI".Mode_auto_actived )
   END_RUNG
   RUNG wire#powerrail
      Contact( "Input_select_auto" )
      Move(in := 2, out1 => "HMI".List_status)
   END_RUNG
   RUNG wire#powerrail
      Contact( "HMI".Mode_manual )
      Contact( "Input_select_manual" )
      R_Coil( "HMI".Mode_auto_actived )
   END_RUNG
   // the same network as SCL:
   IF "HMI".Mode_auto AND "Input_select_auto" THEN "HMI".Mode_auto_actived := TRUE; END_IF;
   IF "Input_select_auto" THEN "HMI".List_status := 2; END_IF;
   IF "HMI".Mode_manual AND "Input_select_manual" THEN "HMI".Mode_auto_actived := FALSE; END_IF;
END_REGION

REGION Network 3
   RUNG wire#powerrail
      Contact( "HMI".Mode_rest )
      Move(in := 0, out1 => "HMI".List_status)
   END_RUNG
   // the same network as SCL:
   IF "HMI".Mode_rest THEN "HMI".List_status := 0; END_IF;
END_REGION

REGION Network 4
   // box feeder
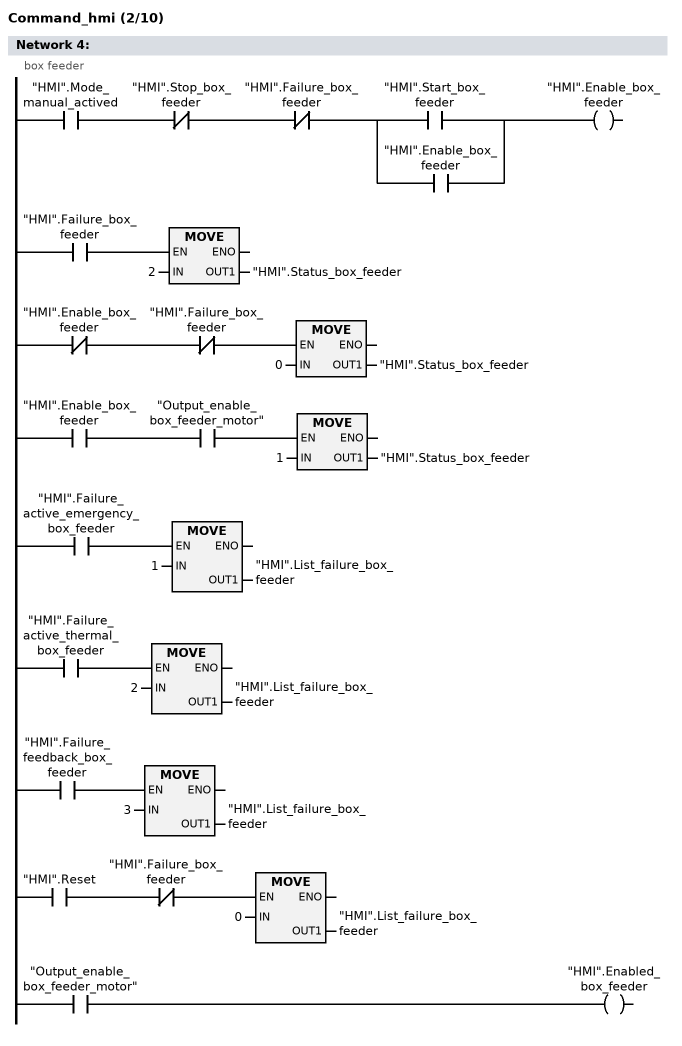
   RUNG wire#powerrail
      Contact( "HMI".Mode_manual_actived )
      I_Contact( "HMI".Stop_box_feeder )
      I_Contact( "HMI".Failure_box_feeder )
      wire#w1
      Contact( "HMI".Start_box_feeder )
      wire#w2
      Coil( "HMI".Enable_box_feeder )
   END_RUNG
   RUNG wire#w1
      Contact( "HMI".Enable_box_feeder )
   END_RUNG wire#w2
   RUNG wire#powerrail
      Contact( "HMI".Failure_box_feeder )
      Move(in := 2, out1 => "HMI".Status_box_feeder)
   END_RUNG
   RUNG wire#powerrail
      I_Contact( "HMI".Enable_box_feeder )
      I_Contact( "HMI".Failure_box_feeder )
      Move(in := 0, out1 => "HMI".Status_box_feeder)
   END_RUNG
   RUNG wire#powerrail
      Contact( "HMI".Enable_box_feeder )
      Contact( "Output_enable_box_feeder_motor" )
      Move(in := 1, out1 => "HMI".Status_box_feeder)
   END_RUNG
   RUNG wire#powerrail
      Contact( "HMI".Failure_active_emergency_box_feeder )
      Move(in := 1, out1 => "HMI".List_failure_box_feeder)
   END_RUNG
   RUNG wire#powerrail
      Contact( "HMI".Failure_active_thermal_box_feeder )
      Move(in := 2, out1 => "HMI".List_failure_box_feeder)
   END_RUNG
   RUNG wire#powerrail
      Contact( "HMI".Failure_feedback_box_feeder )
      Move(in := 3, out1 => "HMI".List_failure_box_feeder)
   END_RUNG
   RUNG wire#powerrail
      Contact( "HMI".Reset )
      I_Contact( "HMI".Failure_box_feeder )
      Move(in := 0, out1 => "HMI".List_failure_box_feeder)
   END_RUNG
   RUNG wire#powerrail
      Contact( "Output_enable_box_feeder_motor" )
      Coil( "HMI".Enabled_box_feeder )
   END_RUNG
   // the same network as SCL:
   "HMI".Enable_box_feeder := "HMI".Mode_manual_actived AND NOT "HMI".Stop_box_feeder AND NOT "HMI".Failure_box_feeder AND ("HMI".Start_box_feeder OR "HMI".Enable_box_feeder);
   IF "HMI".Failure_box_feeder THEN "HMI".Status_box_feeder := 2; END_IF;
   IF NOT "HMI".Enable_box_feeder AND NOT "HMI".Failure_box_feeder THEN "HMI".Status_box_feeder := 0; END_IF;
   IF "HMI".Enable_box_feeder AND "Output_enable_box_feeder_motor" THEN "HMI".Status_box_feeder := 1; END_IF;
   IF "HMI".Failure_active_emergency_box_feeder THEN "HMI".List_failure_box_feeder := 1; END_IF;
   IF "HMI".Failure_active_thermal_box_feeder THEN "HMI".List_failure_box_feeder := 2; END_IF;
   IF "HMI".Failure_feedback_box_feeder THEN "HMI".List_failure_box_feeder := 3; END_IF;
   IF "HMI".Reset AND NOT "HMI".Failure_box_feeder THEN "HMI".List_failure_box_feeder := 0; END_IF;
   "HMI".Enabled_box_feeder := "Output_enable_box_feeder_motor";
END_REGION

REGION Network 5
   // load beld
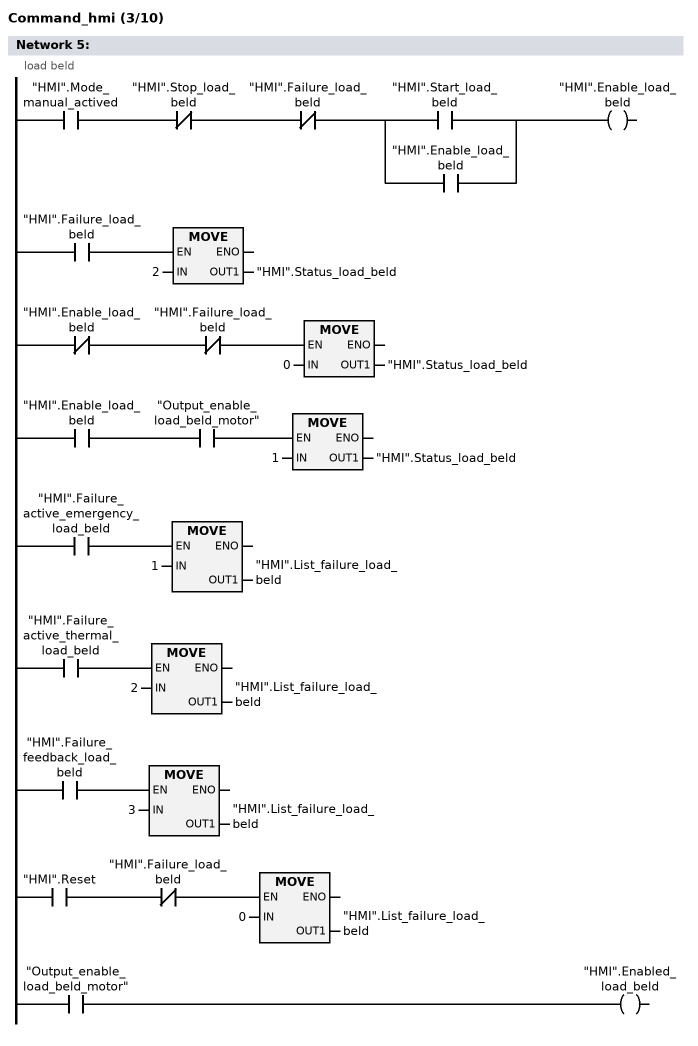
   RUNG wire#powerrail
      Contact( "HMI".Mode_manual_actived )
      I_Contact( "HMI".Stop_load_beld )
      I_Contact( "HMI".Failure_load_beld )
      wire#w1
      Contact( "HMI".Start_load_beld )
      wire#w2
      Coil( "HMI".Enable_load_beld )
   END_RUNG
   RUNG wire#w1
      Contact( "HMI".Enable_load_beld )
   END_RUNG wire#w2
   RUNG wire#powerrail
      Contact( "HMI".Failure_load_beld )
      Move(in := 2, out1 => "HMI".Status_load_beld)
   END_RUNG
   RUNG wire#powerrail
      I_Contact( "HMI".Enable_load_beld )
      I_Contact( "HMI".Failure_load_beld )
      Move(in := 0, out1 => "HMI".Status_load_beld)
   END_RUNG
   RUNG wire#powerrail
      Contact( "HMI".Enable_load_beld )
      Contact( "Output_enable_load_beld_motor" )
      Move(in := 1, out1 => "HMI".Status_load_beld)
   END_RUNG
   RUNG wire#powerrail
      Contact( "HMI".Failure_active_emergency_load_beld )
      Move(in := 1, out1 => "HMI".List_failure_load_beld)
   END_RUNG
   RUNG wire#powerrail
      Contact( "HMI".Failure_active_thermal_load_beld )
      Move(in := 2, out1 => "HMI".List_failure_load_beld)
   END_RUNG
   RUNG wire#powerrail
      Contact( "HMI".Failure_feedback_load_beld )
      Move(in := 3, out1 => "HMI".List_failure_load_beld)
   END_RUNG
   RUNG wire#powerrail
      Contact( "HMI".Reset )
      I_Contact( "HMI".Failure_load_beld )
      Move(in := 0, out1 => "HMI".List_failure_load_beld)
   END_RUNG
   RUNG wire#powerrail
      Contact( "Output_enable_load_beld_motor" )
      Coil( "HMI".Enabled_load_beld )
   END_RUNG
   // the same network as SCL:
   "HMI".Enable_load_beld := "HMI".Mode_manual_actived AND NOT "HMI".Stop_load_beld AND NOT "HMI".Failure_load_beld AND ("HMI".Start_load_beld OR "HMI".Enable_load_beld);
   IF "HMI".Failure_load_beld THEN "HMI".Status_load_beld := 2; END_IF;
   IF NOT "HMI".Enable_load_beld AND NOT "HMI".Failure_load_beld THEN "HMI".Status_load_beld := 0; END_IF;
   IF "HMI".Enable_load_beld AND "Output_enable_load_beld_motor" THEN "HMI".Status_load_beld := 1; END_IF;
   IF "HMI".Failure_active_emergency_load_beld THEN "HMI".List_failure_load_beld := 1; END_IF;
   IF "HMI".Failure_active_thermal_load_beld THEN "HMI".List_failure_load_beld := 2; END_IF;
   IF "HMI".Failure_feedback_load_beld THEN "HMI".List_failure_load_beld := 3; END_IF;
   IF "HMI".Reset AND NOT "HMI".Failure_load_beld THEN "HMI".List_failure_load_beld := 0; END_IF;
   "HMI".Enabled_load_beld := "Output_enable_load_beld_motor";
END_REGION

REGION Network 6
   // elevator
